# B&R Automation Studio project AutomatedPongGame (part 3)

#### testSet_FieldMotor_Disabled.c
```c
/********************************************************************
 * COPYRIGHT - MyAutoMation-IT
 ********************************************************************
 * Author: Raivo Berends
 ********************************************************************/

#include <bur/plctypes.h>

#ifdef _DEFAULT_INCLUDES
#include <AsDefault.h>
#endif

#include "UnitTest.h"
#include "Library.h"
#include "CommonTypes.h"
#include <string.h>

_SETUP_TEST(void)
{
	FieldMotorFB.FieldMotor = &FieldMotorStruct;
	memset(	FieldMotorFB.FieldMotor, 0, sizeof(*FieldMotorFB.FieldMotor));
	FieldMotorFB.FieldMotor->STS.StateInt = STATE_DISABLED;

	TEST_DONE;
}

_TEST test_Disabled_AllOutputsOff(void)
{
	FB_FieldMotor(&FieldMotorFB);

	TEST_ASSERT_EQUAL_INT(0, FieldMotorFB.FieldMotor->CS.Power);
	TEST_ASSERT_EQUAL_INT(0, FieldMotorFB.FieldMotor->CS.Home);
	TEST_ASSERT_EQUAL_INT(0, FieldMotorFB.FieldMotor->CS.MoveJogNeg);
	TEST_ASSERT_EQUAL_INT(0, FieldMotorFB.FieldMotor->CS.MoveJogPos);
	TEST_ASSERT_EQUAL_INT(0, FieldMotorFB.FieldMotor->CS.MoveAbsolute);

	TEST_DONE;
}

_TEST test_Disabled_StatusFlags(void)
{
	FB_FieldMotor(&FieldMotorFB);

	TEST_ASSERT_EQUAL_INT(1, FieldMotorFB.FieldMotor->STS.Disabled);
	TEST_ASSERT_EQUAL_INT(0, FieldMotorFB.FieldMotor->STS.Initializing);
	TEST_ASSERT_EQUAL_INT(0, FieldMotorFB.FieldMotor->STS.Running);
	TEST_ASSERT_EQUAL_INT(0, FieldMotorFB.FieldMotor->STS.Idle);

	TEST_DONE;
}

_TEST test_Disabled_InternalStateReset(void)
{
	FB_FieldMotor(&FieldMotorFB);

	TEST_ASSERT_EQUAL_INT(0, FieldMotorFB.FieldMotor->STS.EndButtonHit);
	TEST_ASSERT_EQUAL_INT(0, FieldMotorFB.FieldMotor->STS.TimerStarted);
	TEST_ASSERT_EQUAL_INT(0, FieldMotorFB.FieldMotor->STS.TimerEnded);
	TEST_ASSERT_EQUAL_INT(0, FieldMotorFB.FieldMotor->STS.ReferencePosition);
	TEST_ASSERT_EQUAL_INT(0, FieldMotorFB.FieldMotor->STS.AtTargetPosition);

	TEST_DONE;
}

_TEST test_Disabled_NoTransitionWithoutInit(void)
{
	FieldMotorFB.FieldMotor->CS.Initialize = 0;

	FB_FieldMotor(&FieldMotorFB);

	TEST_ASSERT_EQUAL_INT(STATE_DISABLED, FieldMotorFB.FieldMotor->STS.StateInt);

	TEST_DONE;
}

_TEST test_Disabled_TransitionsToInitializing(void)
{
	FieldMotorFB.FieldMotor->CS.Initialize = 1;
	FieldMotorFB.FieldMotor->STS.AlarmActive = 0;
	FieldMotorFB.FieldMotor->STS.Interlocked = 0;

	FB_FieldMotor(&FieldMotorFB);

	TEST_ASSERT_EQUAL_INT(STATE_INITIALIZING, FieldMotorFB.FieldMotor->STS.StateInt);

	TEST_DONE;
}

_TEST test_Disabled_BlockedByAlarm(void)
{
	FieldMotorFB.FieldMotor->CS.Initialize = 1;
	FieldMotorFB.FieldMotor->STS.AlarmActive = 1;

	FB_FieldMotor(&FieldMotorFB);

	TEST_ASSERT_EQUAL_INT(STATE_DISABLED, FieldMotorFB.FieldMotor->STS.StateInt);

	TEST_DONE;
}

_TEST test_Disabled_BlockedByInterlock(void)
{
	FieldMotorFB.FieldMotor->CS.Initialize = 1;
	FieldMotorFB.FieldMotor->STS.Interlocked = 1;

	FB_FieldMotor(&FieldMotorFB);

	TEST_ASSERT_EQUAL_INT(STATE_DISABLED, FieldMotorFB.FieldMotor->STS.StateInt);

	TEST_DONE;
}
/*
B+R UnitTest: This is generated code.
Do not edit! Do not move!
Description: UnitTest Testprogramm infrastructure (TestSet).
LastUpdated: 2026-05-01 12:38:40Z
By B+R UnitTest Helper Version: 2.0.2.35
*/
UNITTEST_FIXTURES(fixtures)
{
	new_TestFixture("test_Disabled_AllOutputsOff", test_Disabled_AllOutputsOff),
	new_TestFixture("test_Disabled_StatusFlags", test_Disabled_StatusFlags),
	new_TestFixture("test_Disabled_InternalStateReset", test_Disabled_InternalStateReset),
	new_TestFixture("test_Disabled_NoTransitionWithoutInit", test_Disabled_NoTransitionWithoutInit),
	new_TestFixture("test_Disabled_TransitionsToInitializing", test_Disabled_TransitionsToInitializing),
	new_TestFixture("test_Disabled_BlockedByAlarm", test_Disabled_BlockedByAlarm),
	new_TestFixture("test_Disabled_BlockedByInterlock", test_Disabled_BlockedByInterlock),
};

UNITTEST_CALLER_COMPLETE_EXPLICIT(testSet_FieldMotor_Disabled, "testSet_FieldMotor_Disabled", setupTest, 0, fixtures, 0, 0, 0);
```

#### testSet_FieldMotor_Initializing.c
```c
/********************************************************************
 * COPYRIGHT - MyAutoMation-IT
 ********************************************************************
 * Author: Raivo Berends
 ********************************************************************/

#include <bur/plctypes.h>

#ifdef _DEFAULT_INCLUDES
#include <AsDefault.h>
#endif

#include "UnitTest.h"
#include "Library.h"
#include "CommonTypes.h"
#include <string.h>

#define ENDBUTTON_BITMASK 0x4

_SETUP_TEST(void)
{
	FieldMotorFB.FieldMotor = &FieldMotorStruct;
	memset(FieldMotorFB.FieldMotor, 0, sizeof(*FieldMotorFB.FieldMotor));
	FieldMotorFB.digitalInput = 0;
	FieldMotorFB.FieldMotor->STS.StateInt = STATE_INITIALIZING;

	TEST_DONE;
}

_TEST test_Initializing_SetsPowerAndParameters(void)
{
	FB_FieldMotor(&FieldMotorFB);

	TEST_ASSERT_EQUAL_INT(1, FieldMotorFB.FieldMotor->CS.Power);
	TEST_ASSERT_EQUAL_INT(0, FieldMotorFB.FieldMotor->CS.Stop);

	TEST_ASSERT_EQUAL_INT(MAX_ACC_DEC, FieldMotorFB.FieldMotor->PAR.Acceleration);
	TEST_ASSERT_EQUAL_INT(MAX_ACC_DEC, FieldMotorFB.FieldMotor->PAR.Deceleration);

	TEST_DONE;
}

_TEST test_Initializing_StartsHomingSequence(void)
{
	FieldMotorFB.digitalInput = ENDBUTTON_BITMASK;
	FieldMotorFB.FieldMotor->STS.EndButtonHit = 0;

	FB_FieldMotor(&FieldMotorFB);

	TEST_ASSERT_EQUAL_INT(1, FieldMotorFB.FieldMotor->CS.Home);
	TEST_ASSERT_EQUAL_INT(1, FieldMotorFB.FieldMotor->STS.TimerStarted);

	TEST_DONE;
}

_TEST test_Initializing_EndButtonHit_TriggersCentering(void)
{
	FieldMotorFB.digitalInput = 0;
	FieldMotorFB.FieldMotor->STS.EndButtonHit = 0;

	FB_FieldMotor(&FieldMotorFB);

	TEST_ASSERT_EQUAL_INT(1, FieldMotorFB.FieldMotor->STS.EndButtonHit);
	TEST_ASSERT_EQUAL_INT(1, FieldMotorFB.FieldMotor->CS.Home);
	TEST_ASSERT_EQUAL_INT(1, FieldMotorFB.FieldMotor->CS.SetCenterPoint);

	TEST_DONE;
}

_TEST test_Initializing_TransitionsToIdle(void)
{
	FieldMotorFB.FieldMotor->STS.EndButtonHit = 1;
	FieldMotorFB.FieldMotor->STS.AtTargetPosition = 1;

	FB_FieldMotor(&FieldMotorFB);

	TEST_ASSERT_EQUAL_INT(STATE_IDLE, FieldMotorFB.FieldMotor->STS.StateInt);

	TEST_DONE;
}

_TEST test_Initializing_BlockedByAlarm(void)
{
	FieldMotorFB.FieldMotor->STS.EndButtonHit = 1;
	FieldMotorFB.FieldMotor->STS.AtTargetPosition = 1;
	FieldMotorFB.FieldMotor->STS.AlarmActive = 1;

	FB_FieldMotor(&FieldMotorFB);

	TEST_ASSERT_EQUAL_INT(STATE_INITIALIZING, FieldMotorFB.FieldMotor->STS.StateInt);

	TEST_DONE;
}

_TEST test_Initializing_BlockedByInterlock(void)
{
	FieldMotorFB.FieldMotor->STS.EndButtonHit = 1;
	FieldMotorFB.FieldMotor->STS.AtTargetPosition = 1;
	FieldMotorFB.FieldMotor->STS.Interlocked = 1;

	FB_FieldMotor(&FieldMotorFB);

	TEST_ASSERT_EQUAL_INT(STATE_INITIALIZING, FieldMotorFB.FieldMotor->STS.StateInt);

	TEST_DONE;
}
/*
B+R UnitTest: This is generated code.
Do not edit! Do not move!
Description: UnitTest Testprogramm infrastructure (TestSet).
LastUpdated: 2026-05-01 13:01:47Z
By B+R UnitTest Helper Version: 2.0.2.35
*/
UNITTEST_FIXTURES(fixtures)
{
	new_TestFixture("test_Initializing_SetsPowerAndParameters", test_Initializing_SetsPowerAndParameters),
	new_TestFixture("test_Initializing_StartsHomingSequence", test_Initializing_StartsHomingSequence),
	new_TestFixture("test_Initializing_EndButtonHit_TriggersCentering", test_Initializing_EndButtonHit_TriggersCentering),
	new_TestFixture("test_Initializing_TransitionsToIdle", test_Initializing_TransitionsToIdle),
	new_TestFixture("test_Initializing_BlockedByAlarm", test_Initializing_BlockedByAlarm),
	new_TestFixture("test_Initializing_BlockedByInterlock", test_Initializing_BlockedByInterlock),
};

UNITTEST_CALLER_COMPLETE_EXPLICIT(testSet_FieldMotor_Initializing, "testSet_FieldMotor_Initializing", setupTest, 0, fixtures, 0, 0, 0);
```

#### testSet_FieldMotor_Idle.c
```c
/********************************************************************
 * COPYRIGHT - MyAutoMation-IT
 ********************************************************************
 * Author: Raivo Berends
 ********************************************************************/

#include <bur/plctypes.h>

#ifdef _DEFAULT_INCLUDES
#include <AsDefault.h>
#endif

#include "UnitTest.h"
#include "Library.h"
#include "CommonTypes.h"
#include <string.h>

_SETUP_TEST(void)
{
	FieldMotorFB.FieldMotor = &FieldMotorStruct;
	memset(	FieldMotorFB.FieldMotor, 0, sizeof(*FieldMotorFB.FieldMotor));
	FieldMotorFB.FieldMotor->STS.StateInt = STATE_IDLE;

	TEST_DONE;
}

_TEST test_Idle_AllOutputsOff(void)
{
	FB_FieldMotor(&FieldMotorFB);

	TEST_ASSERT_EQUAL_INT(0, FieldMotorFB.FieldMotor->CS.MoveAbsolute);
	TEST_ASSERT_EQUAL_INT(0, FieldMotorFB.FieldMotor->CS.MoveJogNeg);
	TEST_ASSERT_EQUAL_INT(0, FieldMotorFB.FieldMotor->CS.MoveJogPos);
	TEST_ASSERT_EQUAL_INT(0, FieldMotorFB.FieldMotor->CS.Power);

	TEST_DONE;
}

_TEST test_Idle_StatusFlags(void)
{
	FB_FieldMotor(&FieldMotorFB);

	TEST_ASSERT_EQUAL_INT(1, FieldMotorFB.FieldMotor->STS.Idle);
	TEST_ASSERT_EQUAL_INT(0, FieldMotorFB.FieldMotor->STS.Initializing);
	TEST_ASSERT_EQUAL_INT(0, FieldMotorFB.FieldMotor->STS.Running);

	TEST_DONE;
}

_TEST test_Idle_NoTransitionWithoutStart(void)
{
	FieldMotorFB.FieldMotor->CS.Start = 0;

	FB_FieldMotor(&FieldMotorFB);

	TEST_ASSERT_EQUAL_INT(STATE_IDLE, FieldMotorFB.FieldMotor->STS.StateInt);

	TEST_DONE;
}

_TEST test_Idle_TransitionToRunning(void)
{
	FieldMotorFB.FieldMotor->CS.Start = 1;

	FB_FieldMotor(&FieldMotorFB);

	TEST_ASSERT_EQUAL_INT(STATE_RUNNING, FieldMotorFB.FieldMotor->STS.StateInt);

	TEST_DONE;
}

_TEST test_Idle_BlockedByAlarm(void)
{
	FieldMotorFB.FieldMotor->CS.Start = 1;
	FieldMotorFB.FieldMotor->STS.AlarmActive = 1;

	FB_FieldMotor(&FieldMotorFB);

	TEST_ASSERT_EQUAL_INT(STATE_IDLE, FieldMotorFB.FieldMotor->STS.StateInt);

	TEST_DONE;
}

_TEST test_Idle_BlockedByInterlock(void)
{
	FieldMotorFB.FieldMotor->CS.Start = 1;
	FieldMotorFB.FieldMotor->STS.Interlocked = 1;

	FB_FieldMotor(&FieldMotorFB);

	TEST_ASSERT_EQUAL_INT(STATE_IDLE, FieldMotorFB.FieldMotor->STS.StateInt);

	TEST_DONE;
}
/*
B+R UnitTest: This is generated code.
Do not edit! Do not move!
Description: UnitTest Testprogramm infrastructure (TestSet).
LastUpdated: 2026-05-07 09:05:51Z
By B+R UnitTest Helper Version: 2.0.2.35
*/
UNITTEST_FIXTURES(fixtures)
{
	new_TestFixture("test_Idle_AllOutputsOff", test_Idle_AllOutputsOff),
	new_TestFixture("test_Idle_StatusFlags", test_Idle_StatusFlags),
	new_TestFixture("test_Idle_NoTransitionWithoutStart", test_Idle_NoTransitionWithoutStart),
	new_TestFixture("test_Idle_TransitionToRunning", test_Idle_TransitionToRunning),
	new_TestFixture("test_Idle_BlockedByAlarm", test_Idle_BlockedByAlarm),
	new_TestFixture("test_Idle_BlockedByInterlock", test_Idle_BlockedByInterlock),
};

UNITTEST_CALLER_COMPLETE_EXPLICIT(testSet_FieldMotor_Idle, "testSet_FieldMotor_Idle", setupTest, 0, fixtures, 0, 0, 0);
```

#### testSet_FieldMotor_Running.c
```c
/********************************************************************
 * COPYRIGHT - MyAutoMation-IT
 ********************************************************************
 * Author: Raivo Berends
 ********************************************************************/

#include <bur/plctypes.h>

#ifdef _DEFAULT_INCLUDES
#include <AsDefault.h>
#endif

#include "UnitTest.h"
#include "Library.h"
#include "CommonTypes.h"
#include <string.h>

_SETUP_TEST(void)
{
	FieldMotorFB.FieldMotor = &FieldMotorStruct;
	memset(	FieldMotorFB.FieldMotor, 0, sizeof(*FieldMotorFB.FieldMotor));
	FieldMotorFB.FieldMotor->STS.StateInt = STATE_RUNNING;

	TEST_DONE;
}

_TEST Test_Running_SetsRunningAndPower(void)
{
	FB_FieldMotor(&FieldMotorFB);

	TEST_ASSERT_EQUAL_INT(1, FieldMotorFB.FieldMotor->STS.Running);
	TEST_ASSERT_EQUAL_INT(1, FieldMotorFB.FieldMotor->CS.Power);
	TEST_ASSERT_EQUAL_INT(0, FieldMotorFB.FieldMotor->STS.Idle);

	TEST_DONE;
}

_TEST Test_Running_ResetsMovementCommands(void)
{
	FieldMotorFB.FieldMotor->STS.AutoActive = 0;

	FieldMotorFB.FieldMotor->CS.MoveAbsolute = 1;
	FieldMotorFB.FieldMotor->CS.MoveJogNeg = 1;
	FieldMotorFB.FieldMotor->CS.MoveJogPos = 1;

	FB_FieldMotor(&FieldMotorFB);

	TEST_ASSERT_EQUAL_INT(0, FieldMotorFB.FieldMotor->CS.MoveAbsolute);
	TEST_ASSERT_EQUAL_INT(0, FieldMotorFB.FieldMotor->CS.MoveJogNeg);
	TEST_ASSERT_EQUAL_INT(0, FieldMotorFB.FieldMotor->CS.MoveJogPos);

	TEST_DONE;
}

_TEST Test_Running_IncreaseJogSpeed(void)
{
	FieldMotorFB.FieldMotor->STS.AutoActive = 0;

	FieldMotorFB.FieldMotor->PAR.JogVelocity = 10;
	FieldMotorFB.FieldMotor->HMI.IncreaseJogSpeed = 1;

	FB_FieldMotor(&FieldMotorFB);

	TEST_ASSERT_EQUAL_INT(11, FieldMotorFB.FieldMotor->PAR.JogVelocity);

	TEST_DONE;
}

_TEST Test_Running_MaxJogSpeedLimit(void)
{
	FieldMotorFB.FieldMotor->STS.AutoActive = 0;

	FieldMotorFB.FieldMotor->PAR.JogVelocity = MAX_VELOCITY;
	FieldMotorFB.FieldMotor->HMI.IncreaseJogSpeed = 1;

	FB_FieldMotor(&FieldMotorFB);

	TEST_ASSERT_EQUAL_INT(MAX_VELOCITY, FieldMotorFB.FieldMotor->PAR.JogVelocity);

	TEST_DONE;
}

_TEST Test_Running_DecreaseJogSpeed(void)
{
	FieldMotorFB.FieldMotor->STS.AutoActive = 0;

	FieldMotorFB.FieldMotor->PAR.JogVelocity = 1000;
	FieldMotorFB.FieldMotor->HMI.DecreaseJogSpeed = 1;

	FB_FieldMotor(&FieldMotorFB);

	TEST_ASSERT_EQUAL_INT(999, FieldMotorFB.FieldMotor->PAR.JogVelocity);

	TEST_DONE;
}

_TEST Test_Running_MinJogSpeedLimit(void)
{
	FieldMotorFB.FieldMotor->STS.AutoActive = 0;

	FieldMotorFB.FieldMotor->PAR.JogVelocity = MIN_VELOCITY;
	FieldMotorFB.FieldMotor->HMI.DecreaseJogSpeed = 1;

	FB_FieldMotor(&FieldMotorFB);

	TEST_ASSERT_EQUAL_INT(MIN_VELOCITY, FieldMotorFB.FieldMotor->PAR.JogVelocity);

	TEST_DONE;
}

_TEST Test_Running_EndButtonStopsPositiveMovement(void)
{
	FieldMotorFB.digitalInput = !ENDBUTTON_BITMASK_FIELD;

	FieldMotorFB.FieldMotor->CS.MoveJogPos = 1;
	FieldMotorFB.FieldMotor->HMI.MoveJogPos = 1;
	FieldMotorFB.FieldMotor->CS.MoveAbsolute = 1;

	FB_FieldMotor(&FieldMotorFB);

	TEST_ASSERT_EQUAL_INT(0, FieldMotorFB.FieldMotor->CS.MoveJogPos);
	TEST_ASSERT_EQUAL_INT(0, FieldMotorFB.FieldMotor->HMI.MoveJogPos);
	TEST_ASSERT_EQUAL_INT(0, FieldMotorFB.FieldMotor->CS.MoveAbsolute);

	TEST_DONE;
}

_TEST Test_Running_StopGameTransitionsToStopping(void)
{
	FieldMotorFB.FieldMotor->CS.StopGame = 1;
	FieldMotorFB.FieldMotor->STS.AlarmActive = 0;
	FieldMotorFB.FieldMotor->STS.Interlocked = 0;

	FB_FieldMotor(&FieldMotorFB);

	TEST_ASSERT_EQUAL_INT(STATE_STOPPING, FieldMotorFB.FieldMotor->STS.StateInt);

	TEST_DONE;
}

_TEST Test_Running_StopBlockedByInterlock(void)
{
	FieldMotorFB.FieldMotor->CS.StopGame = 1;
	FieldMotorFB.FieldMotor->STS.Interlocked = 1;

	FB_FieldMotor(&FieldMotorFB);

	TEST_ASSERT_EQUAL_INT(STATE_RUNNING, FieldMotorFB.FieldMotor->STS.StateInt);

	TEST_DONE;
}

_TEST Test_Running_StandStillDetection(void)
{
	FieldMotorFB.FieldMotor->STS.ActVelocity = 0;

	FB_FieldMotor(&FieldMotorFB);

	TEST_ASSERT_EQUAL_INT(1, FieldMotorFB.FieldMotor->STS.StandStill);
	TEST_ASSERT_EQUAL_INT(0, FieldMotorFB.FieldMotor->STS.Moving);

	TEST_DONE;
}

_TEST Test_Running_MovingDetection(void)
{
	FieldMotorFB.FieldMotor->STS.ActVelocity = 100;

	FB_FieldMotor(&FieldMotorFB);

	TEST_ASSERT_EQUAL_INT(0, FieldMotorFB.FieldMotor->STS.StandStill);
	TEST_ASSERT_EQUAL_INT(1, FieldMotorFB.FieldMotor->STS.Moving);

	TEST_DONE;
}

_TEST Test_Running_XorMoveJogPos(void)
{
	FieldMotorFB.FieldMotor->CS.MoveJogPos = 0;
	FieldMotorFB.FieldMotor->HMI.MoveJogPos = 1;
	FieldMotorFB.digitalInput = ENDBUTTON_BITMASK_FIELD;

	FB_FieldMotor(&FieldMotorFB);

	TEST_ASSERT_EQUAL_INT(1, FieldMotorFB.FieldMotor->IO.MoveJogPos);

	TEST_DONE;
}

_TEST Test_Running_XorMoveJogPosBothHigh(void)
{
	FieldMotorFB.FieldMotor->CS.MoveJogPos = 1;
	FieldMotorFB.FieldMotor->HMI.MoveJogPos = 1;
	FieldMotorFB.digitalInput = ENDBUTTON_BITMASK_FIELD;

	FB_FieldMotor(&FieldMotorFB);

	TEST_ASSERT_EQUAL_INT(1, FieldMotorFB.FieldMotor->IO.MoveJogPos);

	TEST_DONE;
}

_TEST Test_Running_AlarmSourcePropagation(void)
{
	FieldMotorFB.FieldMotor->ALM.MotorError = 1;

	FB_FieldMotor(&FieldMotorFB);

	TEST_ASSERT_EQUAL_INT(1, FieldMotorFB.FieldMotor->STS.AlarmActive);

	TEST_DONE;
}

/*
B+R UnitTest: This is generated code.
Do not edit! Do not move!
Description: UnitTest Testprogramm infrastructure (TestSet).
LastUpdated: 2026-05-19 08:31:48Z
By B+R UnitTest Helper Version: 2.0.2.35
*/
UNITTEST_FIXTURES(fixtures)
{
	new_TestFixture("Test_Running_SetsRunningAndPower", Test_Running_SetsRunningAndPower),
	new_TestFixture("Test_Running_ResetsMovementCommands", Test_Running_ResetsMovementCommands),
	new_TestFixture("Test_Running_IncreaseJogSpeed", Test_Running_IncreaseJogSpeed),
	new_TestFixture("Test_Running_MaxJogSpeedLimit", Test_Running_MaxJogSpeedLimit),
	new_TestFixture("Test_Running_DecreaseJogSpeed", Test_Running_DecreaseJogSpeed),
	new_TestFixture("Test_Running_MinJogSpeedLimit", Test_Running_MinJogSpeedLimit),
	new_TestFixture("Test_Running_EndButtonStopsPositiveMovement", Test_Running_EndButtonStopsPositiveMovement),
	new_TestFixture("Test_Running_StopGameTransitionsToStopping", Test_Running_StopGameTransitionsToStopping),
	new_TestFixture("Test_Running_StopBlockedByInterlock", Test_Running_StopBlockedByInterlock),
	new_TestFixture("Test_Running_StandStillDetection", Test_Running_StandStillDetection),
	new_TestFixture("Test_Running_MovingDetection", Test_Running_MovingDetection),
	new_TestFixture("Test_Running_XorMoveJogPos", Test_Running_XorMoveJogPos),
	new_TestFixture("Test_Running_XorMoveJogPosBothHigh", Test_Running_XorMoveJogPosBothHigh),
	new_TestFixture("Test_Running_AlarmSourcePropagation", Test_Running_AlarmSourcePropagation),
};

UNITTEST_CALLER_COMPLETE_EXPLICIT(testSet_FieldMotor_Running, "testSet_FieldMotor_Running", setupTest, 0, fixtures, 0, 0, 0);
```

#### testSet_FieldMotor_Stopping.c
```c
/********************************************************************
 * COPYRIGHT - MyAutoMation-IT
 ********************************************************************
 * Author: Raivo Berends
 ********************************************************************/

#include <bur/plctypes.h>

#ifdef _DEFAULT_INCLUDES
#include <AsDefault.h>
#endif

#include "UnitTest.h"
#include "Library.h"
#include "CommonTypes.h"
#include <string.h>

_SETUP_TEST(void)
{
	FieldMotorFB.FieldMotor = &FieldMotorStruct;
	memset(	FieldMotorFB.FieldMotor, 0, sizeof(*FieldMotorFB.FieldMotor));
	FieldMotorFB.FieldMotor->STS.StateInt = STATE_IDLE;

	TEST_DONE;
}

_TEST Test_Stopping_ResetsStateFlags(void)
{
	FieldMotorFB.FieldMotor->STS.StateInt = STATE_STOPPING;

	FieldMotorFB.FieldMotor->STS.Running = 1;
	FieldMotorFB.FieldMotor->STS.Idle = 1;
	FieldMotorFB.FieldMotor->STS.Initializing = 1;

	FB_FieldMotor(&FieldMotorFB);

	TEST_ASSERT_EQUAL_INT(0, FieldMotorFB.FieldMotor->STS.Running);
	TEST_ASSERT_EQUAL_INT(0, FieldMotorFB.FieldMotor->STS.Idle);
	TEST_ASSERT_EQUAL_INT(0, FieldMotorFB.FieldMotor->STS.Initializing);

	TEST_DONE;
}

_TEST Test_Stopping_StopsAllMovement(void)
{
	FieldMotorFB.FieldMotor->STS.StateInt = STATE_STOPPING;

	FieldMotorFB.FieldMotor->CS.MoveAbsolute = 1;
	FieldMotorFB.FieldMotor->CS.MoveJogNeg = 1;
	FieldMotorFB.FieldMotor->CS.MoveJogPos = 1;

	FB_FieldMotor(&FieldMotorFB);

	TEST_ASSERT_EQUAL_INT(0, FieldMotorFB.FieldMotor->CS.MoveAbsolute);
	TEST_ASSERT_EQUAL_INT(0, FieldMotorFB.FieldMotor->CS.MoveJogNeg);
	TEST_ASSERT_EQUAL_INT(0, FieldMotorFB.FieldMotor->CS.MoveJogPos);

	TEST_DONE;
}

_TEST Test_Stopping_SetsStopCommand(void)
{
	FieldMotorFB.FieldMotor->STS.StateInt = STATE_STOPPING;

	FieldMotorFB.FieldMotor->CS.Stop = 0;

	FB_FieldMotor(&FieldMotorFB);

	TEST_ASSERT_EQUAL_INT(1, FieldMotorFB.FieldMotor->CS.Stop);

	TEST_DONE;
}

_TEST Test_Stopping_TransitionsToDisabled(void)
{
	FieldMotorFB.FieldMotor->STS.StateInt = STATE_STOPPING;

	FieldMotorFB.FieldMotor->STS.StandStill = 1;
	FieldMotorFB.FieldMotor->STS.Interlocked = 0;

	FB_FieldMotor(&FieldMotorFB);

	TEST_ASSERT_EQUAL_INT(STATE_DISABLED, FieldMotorFB.FieldMotor->STS.StateInt);

	TEST_DONE;
}

_TEST Test_Stopping_DoesNotTransitionWhenMoving(void)
{
	FieldMotorFB.FieldMotor->STS.StateInt = STATE_STOPPING;

	FieldMotorFB.FieldMotor->STS.StandStill = 0;
	FieldMotorFB.FieldMotor->STS.Interlocked = 0;

	FB_FieldMotor(&FieldMotorFB);

	TEST_ASSERT_EQUAL_INT(STATE_STOPPING, FieldMotorFB.FieldMotor->STS.StateInt);

	TEST_DONE;
}

_TEST Test_Stopping_DoesNotTransitionWhenInterlocked(void)
{
	FieldMotorFB.FieldMotor->STS.StateInt = STATE_STOPPING;

	FieldMotorFB.FieldMotor->STS.StandStill = 1;
	FieldMotorFB.FieldMotor->STS.Interlocked = 1;

	FB_FieldMotor(&FieldMotorFB);

	TEST_ASSERT_EQUAL_INT(STATE_STOPPING, FieldMotorFB.FieldMotor->STS.StateInt);

	TEST_DONE;
}

_TEST Test_Stopping_UpdatesStopOutput(void)
{
	FieldMotorFB.FieldMotor->STS.StateInt = STATE_STOPPING;

	FB_FieldMotor(&FieldMotorFB);

	TEST_ASSERT_EQUAL_INT(1, FieldMotorFB.FieldMotor->IO.Stop);

	TEST_DONE;
}

/*
B+R UnitTest: This is generated code.
Do not edit! Do not move!
Description: UnitTest Testprogramm infrastructure (TestSet).
LastUpdated: 2026-05-07 09:05:51Z
By B+R UnitTest Helper Version: 2.0.2.35
*/
UNITTEST_FIXTURES(fixtures)
{
	new_TestFixture("Test_Stopping_ResetsStateFlags", Test_Stopping_ResetsStateFlags),
	new_TestFixture("Test_Stopping_StopsAllMovement", Test_Stopping_StopsAllMovement),
	new_TestFixture("Test_Stopping_SetsStopCommand", Test_Stopping_SetsStopCommand),
	new_TestFixture("Test_Stopping_TransitionsToDisabled", Test_Stopping_TransitionsToDisabled),
	new_TestFixture("Test_Stopping_DoesNotTransitionWhenMoving", Test_Stopping_DoesNotTransitionWhenMoving),
	new_TestFixture("Test_Stopping_DoesNotTransitionWhenInterlocked", Test_Stopping_DoesNotTransitionWhenInterlocked),
	new_TestFixture("Test_Stopping_UpdatesStopOutput", Test_Stopping_UpdatesStopOutput),
};

UNITTEST_CALLER_COMPLETE_EXPLICIT(testSet_FieldMotor_Stopping, "testSet_FieldMotor_Stopping", setupTest, 0, fixtures, 0, 0, 0);
```

### Program Logical/UnitTests/UnitTests/Tests_PaddleMotor_C (ANSIC) - Empty template for use with helper tool

#### autoGeneratedFile.c
```c
/*
B+R UnitTest: This is generated code.
Do not edit! Do not move!
Description: UnitTest Testprogramm infrastructure (List of TestSets).
LastUpdated: 2026-05-01 12:04:37Z
By B+R UnitTest Helper Version: 2.0.2.35
*/
#include "UnitTest.h"

UNITTEST_TESTSET_DECLARATION  testSet_PaddleMotor_Disabled;
UNITTEST_TESTSET_DECLARATION  testSet_PaddleMotor_Initializing;
UNITTEST_TESTSET_DECLARATION  testSet_PaddleMotor_Idle;
UNITTEST_TESTSET_DECLARATION  testSet_PaddleMotor_Running;
UNITTEST_TESTSET_DECLARATION  testSet_PaddleMotor_Stopping;

UNITTEST_TESTSET_FIXTURES(utTestSets)
{
	new_TestSet(testSet_PaddleMotor_Disabled),
	new_TestSet(testSet_PaddleMotor_Initializing),
	new_TestSet(testSet_PaddleMotor_Idle),
	new_TestSet(testSet_PaddleMotor_Running),
	new_TestSet(testSet_PaddleMotor_Stopping),
};
UNTITTEST_TESTSET_HANDLER();
```

#### testSet_PaddleMotor_Disabled.c
```c
/********************************************************************
 * COPYRIGHT - MyAutoMation-IT
 ********************************************************************
 * Author: Raivo Berends
 ********************************************************************/

#include <bur/plctypes.h>

#ifdef _DEFAULT_INCLUDES
#include <AsDefault.h>
#endif

#include "UnitTest.h"
#include "Library.h"
#include "CommonTypes.h"
#include <string.h>

_SETUP_TEST(void)
{
	/* TODO:  add code running before test set here */
	PaddleMotorFB.PaddleMotor = &PaddleMotorStruct;
	memset(PaddleMotorFB.PaddleMotor, 0, sizeof(*PaddleMotorFB.PaddleMotor));
	PaddleMotorFB.PaddleMotor->STS.StateInt = STATE_DISABLED;

	TEST_DONE;
}

_TEST test_Disabled_State_DefaultBehavior(void)
{
	PaddleMotorFB.digitalInput = 0;

	// Setting signals that have to be reset
	PaddleMotorFB.PaddleMotor->CS.Power = 1;
	PaddleMotorFB.PaddleMotor->CS.Home = 1;
	PaddleMotorFB.PaddleMotor->CS.MoveJogNeg = 1;
	PaddleMotorFB.PaddleMotor->CS.MoveJogPos = 1;
	PaddleMotorFB.PaddleMotor->CS.MoveAbsolute = 1;

	PaddleMotorFB.PaddleMotor->HMI.MoveJogNeg = 1;
	PaddleMotorFB.PaddleMotor->HMI.MoveJogPos = 1;

	PaddleMotorFB.PaddleMotor->STS.TimerStarted = 1;
	PaddleMotorFB.PaddleMotor->STS.TimerEnded = 1;
	PaddleMotorFB.PaddleMotor->STS.ReferencePosition = 1234;
	PaddleMotorFB.PaddleMotor->STS.ReferenceSet = 1;

	FB_PaddleMotor(&PaddleMotorFB);

	TEST_ASSERT_EQUAL_INT(1, PaddleMotorFB.PaddleMotor->STS.Disabled);

	TEST_ASSERT_EQUAL_INT(0, PaddleMotorFB.PaddleMotor->CS.Power);
	TEST_ASSERT_EQUAL_INT(0, PaddleMotorFB.PaddleMotor->CS.Home);
	TEST_ASSERT_EQUAL_INT(0, PaddleMotorFB.PaddleMotor->CS.MoveJogNeg);
	TEST_ASSERT_EQUAL_INT(0, PaddleMotorFB.PaddleMotor->CS.MoveJogPos);
	TEST_ASSERT_EQUAL_INT(0, PaddleMotorFB.PaddleMotor->CS.MoveAbsolute);

	TEST_ASSERT_EQUAL_INT(0, PaddleMotorFB.PaddleMotor->HMI.MoveJogNeg);
	TEST_ASSERT_EQUAL_INT(0, PaddleMotorFB.PaddleMotor->HMI.MoveJogPos);

	TEST_ASSERT_EQUAL_INT(0, PaddleMotorFB.PaddleMotor->STS.TimerStarted);
	TEST_ASSERT_EQUAL_INT(0, PaddleMotorFB.PaddleMotor->STS.TimerEnded);
	TEST_ASSERT_EQUAL_INT(0, PaddleMotorFB.PaddleMotor->STS.ReferencePosition);
	TEST_ASSERT_EQUAL_INT(0, PaddleMotorFB.PaddleMotor->STS.ReferenceSet);

	TEST_DONE;
}

_TEST test_Disabled_NoInitialize_StaysDisabled(void)
{
	PaddleMotorFB.PaddleMotor->CS.Initialize = 0;
	PaddleMotorFB.PaddleMotor->STS.AlarmActive = 0;
	PaddleMotorFB.PaddleMotor->STS.Interlocked = 0;

	FB_PaddleMotor(&PaddleMotorFB);

	TEST_ASSERT_EQUAL_INT(STATE_DISABLED, PaddleMotorFB.PaddleMotor->STS.StateInt);

	TEST_DONE;
}

_TEST test_Disabled_ToInitializing(void)
{
	PaddleMotorFB.PaddleMotor->CS.Initialize = 1;
	PaddleMotorFB.PaddleMotor->STS.AlarmActive = 0;
	PaddleMotorFB.PaddleMotor->STS.Interlocked = 0;

	FB_PaddleMotor(&PaddleMotorFB);

	TEST_ASSERT_EQUAL_INT(STATE_INITIALIZING, PaddleMotorFB.PaddleMotor->STS.StateInt);

	TEST_DONE;
}

_TEST test_Disabled_NoTransition_WhenAlarm(void)
{
	PaddleMotorFB.PaddleMotor->CS.Initialize = 1;
	PaddleMotorFB.PaddleMotor->STS.AlarmActive = 1;
	PaddleMotorFB.PaddleMotor->STS.Interlocked = 0;

	FB_PaddleMotor(&PaddleMotorFB);

	TEST_ASSERT_EQUAL_INT(STATE_DISABLED, PaddleMotorFB.PaddleMotor->STS.StateInt);

	TEST_DONE;
}

_TEST test_Disabled_NoTransition_WhenInterlocked(void)
{
	PaddleMotorFB.PaddleMotor->CS.Initialize = 1;
	PaddleMotorFB.PaddleMotor->STS.AlarmActive = 0;
	PaddleMotorFB.PaddleMotor->STS.Interlocked = 1;

	FB_PaddleMotor(&PaddleMotorFB);

	TEST_ASSERT_EQUAL_INT(STATE_DISABLED, PaddleMotorFB.PaddleMotor->STS.StateInt);

	TEST_DONE;
}

/*
B+R UnitTest: This is generated code.
Do not edit! Do not move!
Description: UnitTest Testprogramm infrastructure (TestSet).
LastUpdated: 2026-04-20 10:39:20Z
By B+R UnitTest Helper Version: 2.0.2.35
*/
UNITTEST_FIXTURES(fixtures)
{
	new_TestFixture("test_Disabled_State_DefaultBehavior", test_Disabled_State_DefaultBehavior),
	new_TestFixture("test_Disabled_NoInitialize_StaysDisabled", test_Disabled_NoInitialize_StaysDisabled),
	new_TestFixture("test_Disabled_ToInitializing", test_Disabled_ToInitializing),
	new_TestFixture("test_Disabled_NoTransition_WhenAlarm", test_Disabled_NoTransition_WhenAlarm),
	new_TestFixture("test_Disabled_NoTransition_WhenInterlocked", test_Disabled_NoTransition_WhenInterlocked),
};

UNITTEST_CALLER_COMPLETE_EXPLICIT(testSet_PaddleMotor_Disabled, "testSet_PaddleMotor_Disabled", setupTest, 0, fixtures, 0, 0, 0);
```

#### testSet_PaddleMotor_Idle.c
```c
/********************************************************************
 * COPYRIGHT - MyAutoMation-IT
 ********************************************************************
 * Author: Raivo Berends
 ********************************************************************/

#include <bur/plctypes.h>

#ifdef _DEFAULT_INCLUDES
#include <AsDefault.h>
#endif

#include "UnitTest.h"
#include "Library.h"
#include "CommonTypes.h"
#include <string.h>

_SETUP_TEST(void)
{
	PaddleMotorFB.PaddleMotor = &PaddleMotorStruct;
	memset(PaddleMotorFB.PaddleMotor, 0, sizeof(*PaddleMotorFB.PaddleMotor));
	PaddleMotorFB.PaddleMotor->STS.StateInt = STATE_IDLE;

	TEST_DONE;
}

_TEST test_Idle_SetsStatusAndResetsOutputs(void)
{
	PaddleMotorFB.PaddleMotor->STS.Initializing = 1;
	PaddleMotorFB.PaddleMotor->STS.Idle = 0;

	PaddleMotorFB.PaddleMotor->CS.MoveAbsolute = 1;
	PaddleMotorFB.PaddleMotor->CS.MoveJogNeg = 1;
	PaddleMotorFB.PaddleMotor->CS.MoveJogPos = 1;

	PaddleMotorFB.PaddleMotor->HMI.MoveAbsolute = 1;
	PaddleMotorFB.PaddleMotor->HMI.MoveJogNeg = 1;
	PaddleMotorFB.PaddleMotor->HMI.MoveJogPos = 1;

	FB_PaddleMotor(&PaddleMotorFB);

	TEST_ASSERT_EQUAL_INT(0, PaddleMotorFB.PaddleMotor->STS.Initializing);
	TEST_ASSERT_EQUAL_INT(1, PaddleMotorFB.PaddleMotor->STS.Idle);

	TEST_ASSERT_EQUAL_INT(0, PaddleMotorFB.PaddleMotor->CS.MoveAbsolute);
	TEST_ASSERT_EQUAL_INT(0, PaddleMotorFB.PaddleMotor->CS.MoveJogNeg);
	TEST_ASSERT_EQUAL_INT(0, PaddleMotorFB.PaddleMotor->CS.MoveJogPos);

	TEST_ASSERT_EQUAL_INT(0, PaddleMotorFB.PaddleMotor->HMI.MoveAbsolute);
	TEST_ASSERT_EQUAL_INT(0, PaddleMotorFB.PaddleMotor->HMI.MoveJogNeg);
	TEST_ASSERT_EQUAL_INT(0, PaddleMotorFB.PaddleMotor->HMI.MoveJogPos);

	TEST_DONE;
}

_TEST test_Idle_RemainsIdleWithoutStart(void)
{
	PaddleMotorFB.PaddleMotor->CS.Start = 0;

	FB_PaddleMotor(&PaddleMotorFB);

	TEST_ASSERT_EQUAL_INT(STATE_IDLE, PaddleMotorFB.PaddleMotor->STS.StateInt);

	TEST_DONE;
}

_TEST test_Idle_ToRunning(void)
{
	PaddleMotorFB.PaddleMotor->CS.Start = 1;
	PaddleMotorFB.PaddleMotor->STS.AlarmActive = 0;
	PaddleMotorFB.PaddleMotor->STS.Interlocked = 0;

	FB_PaddleMotor(&PaddleMotorFB);

	TEST_ASSERT_EQUAL_INT(STATE_RUNNING, PaddleMotorFB.PaddleMotor->STS.StateInt);

	TEST_DONE;
}

_TEST test_Idle_NoTransitionWhenAlarmActive(void)
{
	PaddleMotorFB.PaddleMotor->CS.Start = 1;
	PaddleMotorFB.PaddleMotor->STS.AlarmActive = 1;
	PaddleMotorFB.PaddleMotor->STS.Interlocked = 0;

	FB_PaddleMotor(&PaddleMotorFB);

	TEST_ASSERT_EQUAL_INT(STATE_IDLE, PaddleMotorFB.PaddleMotor->STS.StateInt);

	TEST_DONE;
}

_TEST test_Idle_NoTransitionWhenInterlocked(void)
{
	PaddleMotorFB.PaddleMotor->CS.Start = 1;
	PaddleMotorFB.PaddleMotor->STS.AlarmActive = 0;
	PaddleMotorFB.PaddleMotor->STS.Interlocked = 1;

	FB_PaddleMotor(&PaddleMotorFB);

	TEST_ASSERT_EQUAL_INT(STATE_IDLE, PaddleMotorFB.PaddleMotor->STS.StateInt);

	TEST_DONE;
}

_TEST test_Idle_IOOutputsRemainZero(void)
{
	PaddleMotorFB.PaddleMotor->CS.MoveJogPos = 0;
	PaddleMotorFB.PaddleMotor->HMI.MoveJogPos = 1;

	PaddleMotorFB.PaddleMotor->CS.MoveJogNeg = 0;
	PaddleMotorFB.PaddleMotor->HMI.MoveJogNeg = 1;

	FB_PaddleMotor(&PaddleMotorFB);

	TEST_ASSERT_EQUAL_INT(0, PaddleMotorFB.PaddleMotor->IO.MoveJogPos);
	TEST_ASSERT_EQUAL_INT(0, PaddleMotorFB.PaddleMotor->IO.MoveJogNeg);

	TEST_DONE;
}

/*
B+R UnitTest: This is generated code.
Do not edit! Do not move!
Description: UnitTest Testprogramm infrastructure (TestSet).
LastUpdated: 2026-05-01 11:23:13Z
By B+R UnitTest Helper Version: 2.0.2.35
*/
UNITTEST_FIXTURES(fixtures)
{
	new_TestFixture("test_Idle_SetsStatusAndResetsOutputs", test_Idle_SetsStatusAndResetsOutputs),
	new_TestFixture("test_Idle_RemainsIdleWithoutStart", test_Idle_RemainsIdleWithoutStart),
	new_TestFixture("test_Idle_ToRunning", test_Idle_ToRunning),
	new_TestFixture("test_Idle_NoTransitionWhenAlarmActive", test_Idle_NoTransitionWhenAlarmActive),
	new_TestFixture("test_Idle_NoTransitionWhenInterlocked", test_Idle_NoTransitionWhenInterlocked),
	new_TestFixture("test_Idle_IOOutputsRemainZero", test_Idle_IOOutputsRemainZero),
};

UNITTEST_CALLER_COMPLETE_EXPLICIT(testSet_PaddleMotor_Idle, "testSet_PaddleMotor_Idle", setupTest, 0, fixtures, 0, 0, 0);
```

#### testSet_PaddleMotor_Initializing.c
```c
/********************************************************************
 * COPYRIGHT - MyAutoMation-IT
 ********************************************************************
 * Author: Raivo Berends
 ********************************************************************/

#include <bur/plctypes.h>

#ifdef _DEFAULT_INCLUDES
#include <AsDefault.h>
#endif

#include "UnitTest.h"
#include "Library.h"
#include "CommonTypes.h"
#include <string.h>

#define MIDDLE_POSITION 1450

_SETUP_TEST(void)
{
	PaddleMotorFB.PaddleMotor = &PaddleMotorStruct;
	memset(PaddleMotorFB.PaddleMotor, 0, sizeof(*PaddleMotorFB.PaddleMotor));
	PaddleMotorFB.PaddleMotor->STS.StateInt = STATE_INITIALIZING;

	TEST_DONE;
}

_TEST test_Initializing_SetsParameters(void)
{
	FB_PaddleMotor(&PaddleMotorFB);

	TEST_ASSERT_EQUAL_INT(1, PaddleMotorFB.PaddleMotor->STS.Initializing);
	TEST_ASSERT_EQUAL_INT(0, PaddleMotorFB.PaddleMotor->STS.Disabled);

	TEST_ASSERT_EQUAL_INT(MAX_ACC_DEC, PaddleMotorFB.PaddleMotor->PAR.Acceleration);
	TEST_ASSERT_EQUAL_INT(MAX_ACC_DEC, PaddleMotorFB.PaddleMotor->PAR.Deceleration);
	TEST_ASSERT_EQUAL_INT(1000, PaddleMotorFB.PaddleMotor->PAR.JogVelocity);
	TEST_ASSERT_EQUAL_INT(1000, PaddleMotorFB.PaddleMotor->PAR.Velocity);

	TEST_ASSERT_EQUAL_INT(1, PaddleMotorFB.PaddleMotor->CS.Power);
	TEST_ASSERT_EQUAL_INT(0, PaddleMotorFB.PaddleMotor->CS.Stop);

	TEST_DONE;
}

_TEST test_Initializing_StartsHoming(void)
{
	PaddleMotorFB.digitalInput = ENDBUTTON_BITMASK_PADDLE; // EndButton = inactive

	PaddleMotorFB.PaddleMotor->STS.EndButtonHit = 0;

	FB_PaddleMotor(&PaddleMotorFB);

	TEST_ASSERT_EQUAL_INT(1, PaddleMotorFB.PaddleMotor->CS.Home);
	TEST_ASSERT_EQUAL_INT(1, PaddleMotorFB.PaddleMotor->STS.TimerStarted);

	TEST_DONE;
}

_TEST test_Initializing_EndButtonHit(void)
{
	PaddleMotorFB.digitalInput = 0x1;

	PaddleMotorFB.PaddleMotor->STS.EndButtonHit = 0;

	FB_PaddleMotor(&PaddleMotorFB);

	TEST_ASSERT_EQUAL_INT(1, PaddleMotorFB.PaddleMotor->STS.EndButtonHit);
	TEST_ASSERT_EQUAL_INT(1, PaddleMotorFB.PaddleMotor->CS.Home);
	TEST_ASSERT_EQUAL_INT(0, PaddleMotorFB.PaddleMotor->CS.MoveJogPos);

	TEST_DONE;
}

_TEST test_Initializing_ToIdle(void)
{
	PaddleMotorFB.PaddleMotor->STS.EndButtonHit = 1;
	PaddleMotorFB.PaddleMotor->STS.TimerEnded = 1;
	PaddleMotorFB.PaddleMotor->STS.ReferenceSet = 1;

	PaddleMotorFB.PaddleMotor->PAR.Position = 3000;
	PaddleMotorFB.PaddleMotor->STS.ActPosition = 3000;

	PaddleMotorFB.PaddleMotor->STS.AlarmActive = 0;
	PaddleMotorFB.PaddleMotor->STS.Interlocked = 0;

	FB_PaddleMotor(&PaddleMotorFB);

	TEST_ASSERT_EQUAL_INT(STATE_IDLE, PaddleMotorFB.PaddleMotor->STS.StateInt);
	TEST_ASSERT_EQUAL_INT(0, PaddleMotorFB.PaddleMotor->CS.MoveAbsolute);

	TEST_DONE;
}

_TEST test_Initializing_ReferencePosition(void)
{
	PaddleMotorFB.PaddleMotor->STS.EndButtonHit = 1;
	PaddleMotorFB.PaddleMotor->STS.TimerEnded = 1;
	PaddleMotorFB.PaddleMotor->STS.ReferenceSet = 0;

	PaddleMotorFB.PaddleMotor->STS.ActPosition = 5000;

	FB_PaddleMotor(&PaddleMotorFB);

	TEST_ASSERT_EQUAL_INT(
		PaddleMotorFB.PaddleMotor->STS.ActPosition + 25,
		PaddleMotorFB.PaddleMotor->STS.ReferencePosition
		);

	TEST_DONE;
}

_TEST test_Initializing_StartMoveAbsolute(void)
{
	PaddleMotorFB.PaddleMotor->STS.EndButtonHit = 1;
	PaddleMotorFB.PaddleMotor->STS.TimerEnded = 1;
	PaddleMotorFB.PaddleMotor->STS.ReferenceSet = 0;

	PaddleMotorFB.PaddleMotor->STS.ActPosition = 4000;

	FB_PaddleMotor(&PaddleMotorFB);

	TEST_ASSERT_EQUAL_INT(1, PaddleMotorFB.PaddleMotor->CS.MoveAbsolute);

	TEST_DONE;
}

_TEST test_Initializing_TargetPosition(void)
{
	PaddleMotorFB.PaddleMotor->STS.EndButtonHit = 1;
	PaddleMotorFB.PaddleMotor->STS.TimerEnded = 1;
	PaddleMotorFB.PaddleMotor->STS.ReferenceSet = 0;

	PaddleMotorFB.PaddleMotor->STS.ActPosition = 5000;

	FB_PaddleMotor(&PaddleMotorFB);

	TEST_ASSERT_EQUAL_INT(
		PaddleMotorFB.PaddleMotor->STS.ReferencePosition - MIDDLE_POSITION,
		PaddleMotorFB.PaddleMotor->PAR.Position
		);

	TEST_DONE;
}
/*
B+R UnitTest: This is generated code.
Do not edit! Do not move!
Description: UnitTest Testprogramm infrastructure (TestSet).
LastUpdated: 2026-05-01 11:41:13Z
By B+R UnitTest Helper Version: 2.0.2.35
*/
UNITTEST_FIXTURES(fixtures)
{
	new_TestFixture("test_Initializing_SetsParameters", test_Initializing_SetsParameters),
	new_TestFixture("test_Initializing_StartsHoming", test_Initializing_StartsHoming),
	new_TestFixture("test_Initializing_EndButtonHit", test_Initializing_EndButtonHit),
	new_TestFixture("test_Initializing_ToIdle", test_Initializing_ToIdle),
	new_TestFixture("test_Initializing_ReferencePosition", test_Initializing_ReferencePosition),
	new_TestFixture("test_Initializing_StartMoveAbsolute", test_Initializing_StartMoveAbsolute),
	new_TestFixture("test_Initializing_TargetPosition", test_Initializing_TargetPosition),
};

UNITTEST_CALLER_COMPLETE_EXPLICIT(testSet_PaddleMotor_Initializing, "testSet_PaddleMotor_Initializing", setupTest, 0, fixtures, 0, 0, 0);
```

#### testSet_PaddleMotor_Running.c
```c
/********************************************************************
 * COPYRIGHT - MyAutoMation-IT
 ********************************************************************
 * Author: Raivo Berends
 ********************************************************************/

#include <bur/plctypes.h>

#ifdef _DEFAULT_INCLUDES
#include <AsDefault.h>
#endif

#include "UnitTest.h"
#include "Library.h"
#include "CommonTypes.h"
#include <string.h>

_SETUP_TEST(void)
{
	PaddleMotorFB.PaddleMotor = &PaddleMotorStruct;

	// volledige reset van alles
	memset(PaddleMotorFB.PaddleMotor, 0, sizeof(*PaddleMotorFB.PaddleMotor));

	// minimale state voor RUNNING tests
	PaddleMotorFB.PaddleMotor->STS.StateInt = STATE_RUNNING;

	TEST_DONE;
}

_TEST test_Running_SetsFlagsCorrectly(void)
{
	PaddleMotorFB.PaddleMotor->STS.Idle = 1;

	FB_PaddleMotor(&PaddleMotorFB);

	TEST_ASSERT_EQUAL_INT(1, PaddleMotorFB.PaddleMotor->STS.Running);
	TEST_ASSERT_EQUAL_INT(0, PaddleMotorFB.PaddleMotor->STS.Idle);

	TEST_DONE;
}

_TEST test_Running_ManualMode_StopsJogging(void)
{
	PaddleMotorFB.PaddleMotor->CS.AutoMode = 0;

	PaddleMotorFB.PaddleMotor->CS.MoveJogNeg = 1;
	PaddleMotorFB.PaddleMotor->CS.MoveJogPos = 1;

	FB_PaddleMotor(&PaddleMotorFB);

	TEST_ASSERT_EQUAL_INT(0, PaddleMotorFB.PaddleMotor->CS.MoveJogNeg);
	TEST_ASSERT_EQUAL_INT(0, PaddleMotorFB.PaddleMotor->CS.MoveJogPos);

	TEST_DONE;
}

_TEST test_Running_IncreaseJogSpeed(void)
{
	PaddleMotorFB.PaddleMotor->CS.AutoMode = 0;

	PaddleMotorFB.PaddleMotor->PAR.JogVelocity = 500;
	PaddleMotorFB.PaddleMotor->HMI.IncreaseJogSpeed = 1;

	FB_PaddleMotor(&PaddleMotorFB);

	TEST_ASSERT_EQUAL_INT(501, PaddleMotorFB.PaddleMotor->PAR.JogVelocity);

	TEST_DONE;
}

_TEST test_Running_DecreaseJogSpeed(void)
{
	PaddleMotorFB.PaddleMotor->CS.AutoMode = 0;

	PaddleMotorFB.PaddleMotor->PAR.JogVelocity = 500;
	PaddleMotorFB.PaddleMotor->HMI.DecreaseJogSpeed = 1;

	FB_PaddleMotor(&PaddleMotorFB);

	TEST_ASSERT_EQUAL_INT(499, PaddleMotorFB.PaddleMotor->PAR.JogVelocity);

	TEST_DONE;
}

_TEST test_Running_IncreaseAccDec(void)
{
	PaddleMotorFB.PaddleMotor->CS.AutoMode = 0;

	PaddleMotorFB.PaddleMotor->PAR.Acceleration = 1000;
	PaddleMotorFB.PaddleMotor->PAR.Deceleration = 1000;

	PaddleMotorFB.PaddleMotor->HMI.IncreaseAccDec = 1;

	FB_PaddleMotor(&PaddleMotorFB);

	TEST_ASSERT_EQUAL_INT(1010, PaddleMotorFB.PaddleMotor->PAR.Acceleration);
	TEST_ASSERT_EQUAL_INT(1010, PaddleMotorFB.PaddleMotor->PAR.Deceleration);

	TEST_DONE;
}

_TEST test_Running_DecreaseAccDec(void)
{
	PaddleMotorFB.PaddleMotor->CS.AutoMode = 0;

	PaddleMotorFB.PaddleMotor->PAR.Acceleration = 2000;
	PaddleMotorFB.PaddleMotor->PAR.Deceleration = 2000;

	PaddleMotorFB.PaddleMotor->HMI.DecreaseAccDec = 1;

	FB_PaddleMotor(&PaddleMotorFB);

	TEST_ASSERT_EQUAL_INT(1990, PaddleMotorFB.PaddleMotor->PAR.Acceleration);
	TEST_ASSERT_EQUAL_INT(1990, PaddleMotorFB.PaddleMotor->PAR.Deceleration);

	TEST_DONE;
}

_TEST test_Running_AutoMode_ResetsHMIInputs(void)
{
	PaddleMotorFB.PaddleMotor->STS.AutoActive = 1;

	PaddleMotorFB.PaddleMotor->HMI.MoveJogNeg = 1;
	PaddleMotorFB.PaddleMotor->HMI.MoveJogPos = 1;
	PaddleMotorFB.PaddleMotor->HMI.MoveAbsolute = 1;

	FB_PaddleMotor(&PaddleMotorFB);

	TEST_ASSERT_EQUAL_INT(0, PaddleMotorFB.PaddleMotor->HMI.MoveJogNeg);
	TEST_ASSERT_EQUAL_INT(0, PaddleMotorFB.PaddleMotor->HMI.MoveJogPos);
	TEST_ASSERT_EQUAL_INT(0, PaddleMotorFB.PaddleMotor->HMI.MoveAbsolute);

	TEST_DONE;
}

_TEST test_Running_LowerLimitProtection(void)
{
	PaddleMotorFB.PaddleMotor->STS.ReferencePosition = 5000;
	PaddleMotorFB.PaddleMotor->STS.ActPosition = 1000;
	PaddleMotorFB.PaddleMotor->STS.ActVelocity = 0;

	FB_PaddleMotor(&PaddleMotorFB);

	TEST_ASSERT_EQUAL_INT(0, PaddleMotorFB.PaddleMotor->CS.MoveJogNeg);

	TEST_DONE;
}

_TEST test_Running_UpperLimitProtection_EndButton(void)
{
	PaddleMotorFB.digitalInput = 0x1;

	FB_PaddleMotor(&PaddleMotorFB);

	TEST_ASSERT_EQUAL_INT(0, PaddleMotorFB.PaddleMotor->CS.MoveJogPos);

	TEST_DONE;
}

_TEST test_Running_UpperLimitProtection_Position(void)
{
	PaddleMotorFB.PaddleMotor->STS.ReferencePosition = 5000;
	PaddleMotorFB.PaddleMotor->STS.ActPosition = 4900;
	PaddleMotorFB.PaddleMotor->STS.ActVelocity = 0;

	FB_PaddleMotor(&PaddleMotorFB);

	TEST_ASSERT_EQUAL_INT(0, PaddleMotorFB.PaddleMotor->CS.MoveJogPos);

	TEST_DONE;
}

_TEST test_Running_StoppingOffset_HighVelocityLimitsMovement(void)
{
	PaddleMotorFB.PaddleMotor->STS.ReferencePosition = 5000;

	// Hoge snelheid ? grote stopping offset
	PaddleMotorFB.PaddleMotor->STS.ActVelocity = 1000;

	// Dicht bij ondergrens
	PaddleMotorFB.PaddleMotor->STS.ActPosition = 2300;

	FB_PaddleMotor(&PaddleMotorFB);

	TEST_ASSERT_EQUAL_INT(0, PaddleMotorFB.PaddleMotor->CS.MoveJogNeg);

	TEST_DONE;
}

_TEST test_Running_LowerLimit_AdjustsTargetPosition(void)
{
	PaddleMotorFB.PaddleMotor->STS.ReferencePosition = 5000;
	PaddleMotorFB.PaddleMotor->STS.ActVelocity = 0;

	// Onder minimum grens
	PaddleMotorFB.PaddleMotor->STS.ActPosition = 1000;

	FB_PaddleMotor(&PaddleMotorFB);

	TEST_ASSERT_EQUAL_INT(PaddleMotorFB.PaddleMotor->STS.ActPosition + 100, PaddleMotorFB.PaddleMotor->PAR.Position);

	TEST_DONE;
}

_TEST test_Running_UpperLimit_AdjustsTargetPosition(void)
{
	PaddleMotorFB.PaddleMotor->STS.ReferencePosition = 5000;
	PaddleMotorFB.PaddleMotor->STS.ActVelocity = 0;

	// Dicht bij bovengrens
	PaddleMotorFB.PaddleMotor->STS.ActPosition = 4950;

	FB_PaddleMotor(&PaddleMotorFB);

	TEST_ASSERT_EQUAL_INT(PaddleMotorFB.PaddleMotor->STS.ReferencePosition - 100, PaddleMotorFB.PaddleMotor->PAR.Position);

	TEST_DONE;
}

_TEST test_Running_EndButton_ForcesStopJogPos(void)
{
	// Activeer endbutton
	PaddleMotorFB.digitalInput = 0x1;

	PaddleMotorFB.PaddleMotor->CS.MoveJogPos = 1;

	FB_PaddleMotor(&PaddleMotorFB);

	TEST_ASSERT_EQUAL_INT(0, PaddleMotorFB.PaddleMotor->CS.MoveJogPos);

	TEST_DONE;
}

_TEST test_Running_StopGame_TransitionsToStopping(void)
{
	PaddleMotorFB.PaddleMotor->CS.StopGame = 1;

	FB_PaddleMotor(&PaddleMotorFB);

	TEST_ASSERT_EQUAL_INT(STATE_STOPPING, PaddleMotorFB.PaddleMotor->STS.StateInt);

	TEST_DONE;
}

_TEST test_Running_StoppingOffset_AffectsUpperLimit(void)
{
	PaddleMotorFB.PaddleMotor->STS.ReferencePosition = 5000;

	// Zonder velocity ? geen offset
	PaddleMotorFB.PaddleMotor->STS.ActVelocity = 0;
	PaddleMotorFB.PaddleMotor->STS.ActPosition = 4900;

	FB_PaddleMotor(&PaddleMotorFB);

	int pos_no_offset = PaddleMotorFB.PaddleMotor->PAR.Position;

	// Reset situatie
	PaddleMotorFB.PaddleMotor->STS.ActVelocity = 1000;
	PaddleMotorFB.PaddleMotor->STS.ActPosition = 4900;

	FB_PaddleMotor(&PaddleMotorFB);

	int pos_with_offset = PaddleMotorFB.PaddleMotor->PAR.Position;

	TEST_ASSERT(pos_with_offset <= pos_no_offset);

	TEST_DONE;
}

/*
B+R UnitTest: This is generated code.
Do not edit! Do not move!
Description: UnitTest Testprogramm infrastructure (TestSet).
LastUpdated: 2026-05-01 12:04:37Z
By B+R UnitTest Helper Version: 2.0.2.35
*/
UNITTEST_FIXTURES(fixtures)
{
	new_TestFixture("test_Running_SetsFlagsCorrectly", test_Running_SetsFlagsCorrectly),
	new_TestFixture("test_Running_ManualMode_StopsJogging", test_Running_ManualMode_StopsJogging),
	new_TestFixture("test_Running_IncreaseJogSpeed", test_Running_IncreaseJogSpeed),
	new_TestFixture("test_Running_DecreaseJogSpeed", test_Running_DecreaseJogSpeed),
	new_TestFixture("test_Running_IncreaseAccDec", test_Running_IncreaseAccDec),
	new_TestFixture("test_Running_DecreaseAccDec", test_Running_DecreaseAccDec),
	new_TestFixture("test_Running_AutoMode_ResetsHMIInputs", test_Running_AutoMode_ResetsHMIInputs),
	new_TestFixture("test_Running_LowerLimitProtection", test_Running_LowerLimitProtection),
	new_TestFixture("test_Running_UpperLimitProtection_EndButton", test_Running_UpperLimitProtection_EndButton),
	new_TestFixture("test_Running_UpperLimitProtection_Position", test_Running_UpperLimitProtection_Position),
	new_TestFixture("test_Running_StoppingOffset_HighVelocityLimitsMovement", test_Running_StoppingOffset_HighVelocityLimitsMovement),
	new_TestFixture("test_Running_LowerLimit_AdjustsTargetPosition", test_Running_LowerLimit_AdjustsTargetPosition),
	new_TestFixture("test_Running_UpperLimit_AdjustsTargetPosition", test_Running_UpperLimit_AdjustsTargetPosition),
	new_TestFixture("test_Running_EndButton_ForcesStopJogPos", test_Running_EndButton_ForcesStopJogPos),
	new_TestFixture("test_Running_StopGame_TransitionsToStopping", test_Running_StopGame_TransitionsToStopping),
	new_TestFixture("test_Running_StoppingOffset_AffectsUpperLimit", test_Running_StoppingOffset_AffectsUpperLimit),
};

UNITTEST_CALLER_COMPLETE_EXPLICIT(testSet_PaddleMotor_Running, "testSet_PaddleMotor_Running", setupTest, 0, fixtures, 0, 0, 0);
```

#### testSet_PaddleMotor_Stopping.c
```c
/********************************************************************
 * COPYRIGHT - MyAutoMation-IT
 ********************************************************************
 * Author: Raivo Berends
 ********************************************************************/

#include <bur/plctypes.h>

#ifdef _DEFAULT_INCLUDES
#include <AsDefault.h>
#endif

#include "UnitTest.h"
#include "Library.h"
#include "CommonTypes.h"
#include <string.h>

_SETUP_TEST(void)
{
	PaddleMotorFB.PaddleMotor = &PaddleMotorStruct;
	memset(PaddleMotorFB.PaddleMotor, 0, sizeof(*PaddleMotorFB.PaddleMotor));
	PaddleMotorFB.PaddleMotor->STS.StateInt = STATE_STOPPING;

	TEST_DONE;
}

_TEST test_Stopping_AllCommandsReset(void)
{
	FB_PaddleMotor(&PaddleMotorFB);

	TEST_ASSERT_EQUAL_INT(0, PaddleMotorFB.PaddleMotor->CS.MoveAbsolute);
	TEST_ASSERT_EQUAL_INT(0, PaddleMotorFB.PaddleMotor->CS.MoveJogNeg);
	TEST_ASSERT_EQUAL_INT(0, PaddleMotorFB.PaddleMotor->CS.MoveJogPos);
	TEST_ASSERT_EQUAL_INT(1, PaddleMotorFB.PaddleMotor->CS.Stop);

	TEST_DONE;
}

_TEST test_Stopping_RemainsInState_WhenNotStandStill(void)
{
	PaddleMotorFB.PaddleMotor->STS.StandStill = 0;
	PaddleMotorFB.PaddleMotor->STS.Interlocked = 0;

	FB_PaddleMotor(&PaddleMotorFB);

	TEST_ASSERT_EQUAL_INT(STATE_STOPPING, PaddleMotorFB.PaddleMotor->STS.StateInt);

	TEST_DONE;
}

_TEST test_Stopping_ToDisabled_WhenStandStill(void)
{
	PaddleMotorFB.PaddleMotor->STS.StandStill = 1;
	PaddleMotorFB.PaddleMotor->STS.Interlocked = 0;

	FB_PaddleMotor(&PaddleMotorFB);

	TEST_ASSERT_EQUAL_INT(STATE_DISABLED, PaddleMotorFB.PaddleMotor->STS.StateInt);

	TEST_DONE;
}

_TEST test_Stopping_NoTransition_WhenInterlocked(void)
{
	PaddleMotorFB.PaddleMotor->STS.StandStill = 1;
	PaddleMotorFB.PaddleMotor->STS.Interlocked = 1;

	FB_PaddleMotor(&PaddleMotorFB);

	TEST_ASSERT_EQUAL_INT(STATE_STOPPING, PaddleMotorFB.PaddleMotor->STS.StateInt);

	TEST_DONE;
}

_TEST test_Stopping_StopSignalAlwaysActive(void)
{
	FB_PaddleMotor(&PaddleMotorFB);

	TEST_ASSERT_EQUAL_INT(1, PaddleMotorFB.PaddleMotor->CS.Stop);

	TEST_DONE;
}

/*
B+R UnitTest: This is generated code.
Do not edit! Do not move!
Description: UnitTest Testprogramm infrastructure (TestSet).
LastUpdated: 2026-05-01 12:04:37Z
By B+R UnitTest Helper Version: 2.0.2.35
*/
UNITTEST_FIXTURES(fixtures)
{
	new_TestFixture("test_Stopping_AllCommandsReset", test_Stopping_AllCommandsReset),
	new_TestFixture("test_Stopping_RemainsInState_WhenNotStandStill", test_Stopping_RemainsInState_WhenNotStandStill),
	new_TestFixture("test_Stopping_ToDisabled_WhenStandStill", test_Stopping_ToDisabled_WhenStandStill),
	new_TestFixture("test_Stopping_NoTransition_WhenInterlocked", test_Stopping_NoTransition_WhenInterlocked),
	new_TestFixture("test_Stopping_StopSignalAlwaysActive", test_Stopping_StopSignalAlwaysActive),
};

UNITTEST_CALLER_COMPLETE_EXPLICIT(testSet_PaddleMotor_Stopping, "testSet_PaddleMotor_Stopping", setupTest, 0, fixtures, 0, 0, 0);
```

#### testSuite.c
```c
/********************************************************************
 * COPYRIGHT --
 ********************************************************************
 * Program: -
 * Author:
 * Created:
 ********************************************************************
 * Test registration and handshake
 ********************************************************************/

#include <bur/plctypes.h>

#ifdef _DEFAULT_INCLUDES
#include <AsDefault.h>
#endif

#include "UnitTest.h"
#include "Library.h"

void _INIT initTestSuite(void)
{
	utInit(&Testsuite);
}

void _CYCLIC cyclicWithTest(void)
{
	utCyclic(&Testsuite);
}

void _EXIT exitTestSuite(void)
{
	utExit(&Testsuite);
}
```

### Package Logical/UnitTests/UnitTests/TestSet_Templates - Multiple variants of valid test sets

### testSet_Template.c
```c
/********************************************************************
 * COPYRIGHT - MyAutoMation-IT
 ********************************************************************
 * Author: Raivo Berends
 ********************************************************************/

#include <bur/plctypes.h>

#ifdef _DEFAULT_INCLUDES
#include <AsDefault.h>
#endif

#include "UnitTest.h"
#include "Library.h"
#include "CommonTypes.h"

_SETUP_TEST(void)
{
	PaddleMotorFB.PaddleMotor = &PaddleMotorStruct;
	PaddleMotorFB.PaddleMotor->STS.StateInt = STATE_IDLE;

	TEST_DONE;
}

_TEST test_Template(void)
{
}

/*
B+R UnitTest: This is generated code.
Do not edit! Do not move!
Description: UnitTest Testprogramm infrastructure (TestSet).
LastUpdated: 2026-05-01 11:23:13Z
By B+R UnitTest Helper Version: 2.0.2.35
*/
UNITTEST_FIXTURES(fixtures)
{
};

UNITTEST_CALLER_COMPLETE_EXPLICIT(testSet_PaddleMotor_Idle, "testSet_Template", setupTest, 0, fixtures, 0, 0, 0);
```

### Program Logical/UnitTests/UnitTests/Tests_BallControl_C (ANSIC)

#### variables.var - Name the suite and add PVs for the program
```iecst
(********************************************************************
 * COPYRIGHT --  MyAutomation-IT
 ********************************************************************
 * Program: Tests_BallControl_C
 * File: variables.var
 * Author: Raivo Berends
 ********************************************************************
 * Local variables of program Tests_BallControl_C
 ********************************************************************)
(*Describe the test*)
VAR
	Testsuite : UtMgrTestSuite := (Name:='BallControl_Tests',Type:=utMgrTEST_TYPE_C);
END_VAR
(*Variables used in the tests*)
VAR
	BallControlFB : FB_BallControl;
	DistanceSensorLeftStruct : UDT_DistanceSensor;
	DistanceSensorMiddleStruct : UDT_DistanceSensor;
	DistanceSensorRightStruct : UDT_DistanceSensor;
	BallControlStruct : UDT_BallControl;
	PaddleMotorStruct : UDT_PaddleMotor;
	ShooterStruct : UDT_Shooter;
END_VAR
```

#### autoGeneratedFile.c - Auto generated code - list of all test sets in the program
```c
/*
B+R UnitTest: This is generated code.
Do not edit! Do not move!
Description: UnitTest Testprogramm infrastructure (List of TestSets).
LastUpdated: 2026-05-07 12:26:03Z
By B+R UnitTest Helper Version: 2.0.2.35
*/
#include "UnitTest.h"

UNITTEST_TESTSET_DECLARATION  testSet_BallControl_Disabled;
UNITTEST_TESTSET_DECLARATION  testSet_BallControl_Initializing;
UNITTEST_TESTSET_DECLARATION  testSet_BallControl_Idle;
UNITTEST_TESTSET_DECLARATION  testSet_BallControl_Running;
UNITTEST_TESTSET_DECLARATION  testSet_BallControl_Stopping;

UNITTEST_TESTSET_FIXTURES(utTestSets)
{
	new_TestSet(testSet_BallControl_Disabled),
	new_TestSet(testSet_BallControl_Initializing),
	new_TestSet(testSet_BallControl_Idle),
	new_TestSet(testSet_BallControl_Running),
	new_TestSet(testSet_BallControl_Stopping),
};
UNTITTEST_TESTSET_HANDLER();
```

#### testSet_BallControl_Disabled.c
```c
/********************************************************************
 * COPYRIGHT - MyAutoMation-IT
 ********************************************************************
 * Author: Raivo Berends
 ********************************************************************/

#include <bur/plctypes.h>

#ifdef _DEFAULT_INCLUDES
#include <AsDefault.h>
#endif

#include "UnitTest.h"
#include "Library.h"
#include "CommonTypes.h"
#include <string.h>

_SETUP_TEST(void)
{
	BallControlFB.BallControl = &BallControlStruct;
	BallControlFB.DistanceSensorLeft = &DistanceSensorLeftStruct;
	BallControlFB.DistanceSensorMiddle = &DistanceSensorMiddleStruct;
	BallControlFB.DistanceSensorRight = &DistanceSensorRightStruct;
	BallControlFB.PaddleMotor = &PaddleMotorStruct;
	BallControlFB.Shooter = &ShooterStruct;

	memset(BallControlFB.BallControl, 0, sizeof(*BallControlFB.BallControl));
	memset(BallControlFB.DistanceSensorLeft, 0, sizeof(*BallControlFB.DistanceSensorLeft));
	memset(BallControlFB.DistanceSensorMiddle, 0, sizeof(*BallControlFB.DistanceSensorMiddle));
	memset(BallControlFB.DistanceSensorRight, 0, sizeof(*BallControlFB.DistanceSensorRight));
	memset(BallControlFB.PaddleMotor, 0, sizeof(*BallControlFB.PaddleMotor));
	memset(BallControlFB.Shooter, 0, sizeof(*BallControlFB.Shooter));

	BallControlFB.BallControl->STS.StateInt = STATE_DISABLED;

	TEST_DONE;
}

_TEST Test_Disabled_ResetsShoot(void)
{
	BallControlFB.BallControl->CS.Shoot = 1;

	FB_BallControl(&BallControlFB);

	TEST_ASSERT_EQUAL_INT(0, BallControlFB.BallControl->CS.Shoot);

	TEST_DONE;
}

_TEST Test_Disabled_IntensityIncrease(void)
{
	BallControlFB.Shooter->HMI.IncreaseIntensity = 1;
	BallControlFB.Shooter->PAR.Intensity = 5;

	FB_BallControl(&BallControlFB);

	TEST_ASSERT(BallControlFB.Shooter->PAR.Intensity > 5);

	TEST_DONE;
}

_TEST Test_Disabled_IntensityDecrease(void)
{
	BallControlFB.Shooter->HMI.DecreaseIntensity = 1;
	BallControlFB.Shooter->PAR.Intensity = 5;

	FB_BallControl(&BallControlFB);

	TEST_ASSERT(BallControlFB.Shooter->PAR.Intensity < 5);

	TEST_DONE;
}

_TEST Test_Disabled_IntensityUpperLimit(void)
{
	BallControlFB.Shooter->HMI.IncreaseIntensity = 1;
	BallControlFB.Shooter->PAR.Intensity = MAX_INTENSITY;

	FB_BallControl(&BallControlFB);

	TEST_ASSERT_EQUAL_INT(MAX_INTENSITY, BallControlFB.Shooter->PAR.Intensity);

	TEST_DONE;
}

_TEST Test_Disabled_IntensityLowerLimit(void)
{
	BallControlFB.Shooter->HMI.DecreaseIntensity = 1;
	BallControlFB.Shooter->PAR.Intensity = MIN_INTENSITY;

	FB_BallControl(&BallControlFB);

	TEST_ASSERT_EQUAL_INT(MIN_INTENSITY, BallControlFB.Shooter->PAR.Intensity);

	TEST_DONE;
}

_TEST Test_Disabled_TransitionsToInitializing(void)
{
	BallControlFB.BallControl->STS.Initializing = 1;

	FB_BallControl(&BallControlFB);

	TEST_ASSERT_EQUAL_INT(STATE_INITIALIZING, BallControlFB.BallControl->STS.StateInt);

	TEST_DONE;
}

_TEST Test_Disabled_NoTransitionWithoutInit(void)
{
	BallControlFB.BallControl->STS.Initializing = 0;

	FB_BallControl(&BallControlFB);

	TEST_ASSERT_EQUAL_INT(STATE_DISABLED, BallControlFB.BallControl->STS.StateInt);

	TEST_DONE;
}

_TEST Test_Disabled_StopsOnlyShootCommand(void)
{
	BallControlFB.BallControl->CS.Shoot = 1;
	BallControlFB.BallControl->CS.AutoMode = 1;

	FB_BallControl(&BallControlFB);

	TEST_ASSERT_EQUAL_INT(0, BallControlFB.BallControl->CS.Shoot);
	TEST_ASSERT_EQUAL_INT(1, BallControlFB.BallControl->CS.AutoMode);

	TEST_DONE;
}

/*
B+R UnitTest: This is generated code.
Do not edit! Do not move!
Description: UnitTest Testprogramm infrastructure (TestSet).
LastUpdated: 2026-05-07 11:56:27Z
By B+R UnitTest Helper Version: 2.0.2.35
*/
UNITTEST_FIXTURES(fixtures)
{
	new_TestFixture("Test_Disabled_ResetsShoot", Test_Disabled_ResetsShoot),
	new_TestFixture("Test_Disabled_IntensityIncrease", Test_Disabled_IntensityIncrease),
	new_TestFixture("Test_Disabled_IntensityDecrease", Test_Disabled_IntensityDecrease),
	new_TestFixture("Test_Disabled_IntensityUpperLimit", Test_Disabled_IntensityUpperLimit),
	new_TestFixture("Test_Disabled_IntensityLowerLimit", Test_Disabled_IntensityLowerLimit),
	new_TestFixture("Test_Disabled_TransitionsToInitializing", Test_Disabled_TransitionsToInitializing),
	new_TestFixture("Test_Disabled_NoTransitionWithoutInit", Test_Disabled_NoTransitionWithoutInit),
	new_TestFixture("Test_Disabled_StopsOnlyShootCommand", Test_Disabled_StopsOnlyShootCommand),
};

UNITTEST_CALLER_COMPLETE_EXPLICIT(testSet_BallControl_Disabled, "testSet_BallControl_Disabled", setupTest, 0, fixtures, 0, 0, 0);
```

#### testSet_BallControl_Initializing.c
```c
/********************************************************************
 * COPYRIGHT - MyAutoMation-IT
 ********************************************************************
 * Author: Raivo Berends
 ********************************************************************/

#include <bur/plctypes.h>

#ifdef _DEFAULT_INCLUDES
#include <AsDefault.h>
#endif

#include "UnitTest.h"
#include "Library.h"
#include "CommonTypes.h"
#include <string.h>

_SETUP_TEST(void)
{
	BallControlFB.BallControl = &BallControlStruct;
	BallControlFB.DistanceSensorLeft = &DistanceSensorLeftStruct;
	BallControlFB.DistanceSensorMiddle = &DistanceSensorMiddleStruct;
	BallControlFB.DistanceSensorRight = &DistanceSensorRightStruct;
	BallControlFB.PaddleMotor = &PaddleMotorStruct;
	BallControlFB.Shooter = &ShooterStruct;

	memset(BallControlFB.BallControl, 0, sizeof(*BallControlFB.BallControl));
	memset(BallControlFB.DistanceSensorLeft, 0, sizeof(*BallControlFB.DistanceSensorLeft));
	memset(BallControlFB.DistanceSensorMiddle, 0, sizeof(*BallControlFB.DistanceSensorMiddle));
	memset(BallControlFB.DistanceSensorRight, 0, sizeof(*BallControlFB.DistanceSensorRight));
	memset(BallControlFB.PaddleMotor, 0, sizeof(*BallControlFB.PaddleMotor));
	memset(BallControlFB.Shooter, 0, sizeof(*BallControlFB.Shooter));

	BallControlFB.BallControl->STS.StateInt = STATE_INITIALIZING;

	TEST_DONE;
}

_TEST Test_Initializing_ResetsStates(void)
{
	BallControlFB.BallControl->STS.PrevShootState = 5;
	BallControlFB.BallControl->STS.ShootState = 10;
	BallControlFB.BallControl->STS.GameOver = 1;
	BallControlFB.BallControl->STS.FirstRun = 0;

	FB_BallControl(&BallControlFB);

	TEST_ASSERT_EQUAL_INT(0, BallControlFB.BallControl->STS.PrevShootState);
	TEST_ASSERT_EQUAL_INT(0, BallControlFB.BallControl->STS.ShootState);
	TEST_ASSERT_EQUAL_INT(0, BallControlFB.BallControl->STS.GameOver);
	TEST_ASSERT_EQUAL_INT(1, BallControlFB.BallControl->STS.FirstRun);

	TEST_DONE;
}

_TEST Test_Initializing_TransitionsToIdle(void)
{
	BallControlFB.BallControl->STS.Idle = 1;

	FB_BallControl(&BallControlFB);

	TEST_ASSERT_EQUAL_INT(STATE_IDLE, BallControlFB.BallControl->STS.StateInt);

	TEST_DONE;
}

_TEST Test_Initializing_NoIdleStaysInState(void)
{;
	BallControlFB.BallControl->STS.Idle = 0;

	FB_BallControl(&BallControlFB);

	TEST_ASSERT_EQUAL_INT(STATE_INITIALIZING, BallControlFB.BallControl->STS.StateInt);

	TEST_DONE;
}

/*
B+R UnitTest: This is generated code.
Do not edit! Do not move!
Description: UnitTest Testprogramm infrastructure (TestSet).
LastUpdated: 2026-05-07 12:20:57Z
By B+R UnitTest Helper Version: 2.0.2.35
*/
UNITTEST_FIXTURES(fixtures)
{
	new_TestFixture("Test_Initializing_ResetsStates", Test_Initializing_ResetsStates),
	new_TestFixture("Test_Initializing_TransitionsToIdle", Test_Initializing_TransitionsToIdle),
	new_TestFixture("Test_Initializing_NoIdleStaysInState", Test_Initializing_NoIdleStaysInState),
};

UNITTEST_CALLER_COMPLETE_EXPLICIT(testSet_BallControl_Initializing, "testSet_BallControl_Initializing", setupTest, 0, fixtures, 0, 0, 0);
```

#### testSet_BallControl_Idle.c
```c
/********************************************************************
 * COPYRIGHT - MyAutoMation-IT
 ********************************************************************
 * Author: Raivo Berends
 ********************************************************************/

#include <bur/plctypes.h>

#ifdef _DEFAULT_INCLUDES
#include <AsDefault.h>
#endif

#include "UnitTest.h"
#include "Library.h"
#include "CommonTypes.h"
#include <string.h>

_SETUP_TEST(void)
{
	BallControlFB.BallControl = &BallControlStruct;
	BallControlFB.DistanceSensorLeft = &DistanceSensorLeftStruct;
	BallControlFB.DistanceSensorMiddle = &DistanceSensorMiddleStruct;
	BallControlFB.DistanceSensorRight = &DistanceSensorRightStruct;
	BallControlFB.PaddleMotor = &PaddleMotorStruct;
	BallControlFB.Shooter = &ShooterStruct;

	memset(BallControlFB.BallControl, 0, sizeof(*BallControlFB.BallControl));
	memset(BallControlFB.DistanceSensorLeft, 0, sizeof(*BallControlFB.DistanceSensorLeft));
	memset(BallControlFB.DistanceSensorMiddle, 0, sizeof(*BallControlFB.DistanceSensorMiddle));
	memset(BallControlFB.DistanceSensorRight, 0, sizeof(*BallControlFB.DistanceSensorRight));
	memset(BallControlFB.PaddleMotor, 0, sizeof(*BallControlFB.PaddleMotor));
	memset(BallControlFB.Shooter, 0, sizeof(*BallControlFB.Shooter));

	BallControlFB.BallControl->STS.StateInt = STATE_IDLE;

	TEST_DONE;
}

_TEST Test_Idle_StaysIdle_WhenNotRunning(void)
{
	BallControlFB.BallControl->STS.Running = 0;

	FB_BallControl(&BallControlFB);

	TEST_ASSERT_EQUAL_INT(STATE_IDLE, BallControlFB.BallControl->STS.StateInt);

	TEST_DONE;
}

_TEST Test_Idle_TransitionsToRunning_WhenRunningTrue(void)
{
	BallControlFB.BallControl->STS.Running = 1;

	FB_BallControl(&BallControlFB);

	TEST_ASSERT_EQUAL_INT(STATE_RUNNING, BallControlFB.BallControl->STS.StateInt);

	TEST_DONE;
}

_TEST Test_Idle_TransitionsOnlyOnRunningTrue(void)
{
	/* cycle 1: not running */
	BallControlFB.BallControl->STS.Running = 0;
	FB_BallControl(&BallControlFB);
	TEST_ASSERT_EQUAL_INT(STATE_IDLE, BallControlFB.BallControl->STS.StateInt);

	/* cycle 2: running becomes true */
	BallControlFB.BallControl->STS.Running = 1;
	FB_BallControl(&BallControlFB);
	TEST_ASSERT_EQUAL_INT(STATE_RUNNING, BallControlFB.BallControl->STS.StateInt);

	TEST_DONE;
}

/*
B+R UnitTest: This is generated code.
Do not edit! Do not move!
Description: UnitTest Testprogramm infrastructure (TestSet).
LastUpdated: 2026-05-07 12:26:03Z
By B+R UnitTest Helper Version: 2.0.2.35
*/
UNITTEST_FIXTURES(fixtures)
{
	new_TestFixture("Test_Idle_StaysIdle_WhenNotRunning", Test_Idle_StaysIdle_WhenNotRunning),
	new_TestFixture("Test_Idle_TransitionsToRunning_WhenRunningTrue", Test_Idle_TransitionsToRunning_WhenRunningTrue),
	new_TestFixture("Test_Idle_TransitionsOnlyOnRunningTrue", Test_Idle_TransitionsOnlyOnRunningTrue),
};

UNITTEST_CALLER_COMPLETE_EXPLICIT(testSet_BallControl_Idle, "testSet_BallControl_Idle", setupTest, 0, fixtures, 0, 0, 0);
```

#### testSet_BallControl_Running.c
```c
/********************************************************************
 * COPYRIGHT - MyAutoMation-IT
 ********************************************************************
 * Author: Raivo Berends
 ********************************************************************/

#include <bur/plctypes.h>

#ifdef _DEFAULT_INCLUDES
#include <AsDefault.h>
#endif

#include "UnitTest.h"
#include "Library.h"
#include "CommonTypes.h"
#include <string.h>

_SETUP_TEST(void)
{
	BallControlFB.BallControl = &BallControlStruct;
	BallControlFB.DistanceSensorLeft = &DistanceSensorLeftStruct;
	BallControlFB.DistanceSensorMiddle = &DistanceSensorMiddleStruct;
	BallControlFB.DistanceSensorRight = &DistanceSensorRightStruct;
	BallControlFB.PaddleMotor = &PaddleMotorStruct;
	BallControlFB.Shooter = &ShooterStruct;

	memset(BallControlFB.BallControl, 0, sizeof(*BallControlFB.BallControl));
	memset(BallControlFB.DistanceSensorLeft, 0, sizeof(*BallControlFB.DistanceSensorLeft));
	memset(BallControlFB.DistanceSensorMiddle, 0, sizeof(*BallControlFB.DistanceSensorMiddle));
	memset(BallControlFB.DistanceSensorRight, 0, sizeof(*BallControlFB.DistanceSensorRight));
	memset(BallControlFB.PaddleMotor, 0, sizeof(*BallControlFB.PaddleMotor));
	memset(BallControlFB.Shooter, 0, sizeof(*BallControlFB.Shooter));

	BallControlFB.BallControl->STS.StateInt = STATE_RUNNING;

	TEST_DONE;
}

_TEST Test_Running_AutoActive_SetsOutputs(void)
{
	BallControlFB.BallControl->STS.AutoActive = 1;

	FB_BallControl(&BallControlFB);

	TEST_ASSERT_EQUAL_INT(0, BallControlFB.PaddleMotor->CS.MoveAbsolute);
	TEST_ASSERT_EQUAL_INT(1, BallControlFB.Shooter->CS.EnableFan);
	TEST_ASSERT_EQUAL_INT(AUTOMODE_VELOCITY, BallControlFB.PaddleMotor->PAR.Velocity);

	TEST_DONE;
}

_TEST Test_Running_WhenAutoInactive_DisablesShoot(void)
{
	BallControlFB.BallControl->STS.AutoActive = 0;

	BallControlFB.BallControl->CS.Shoot = 1;

	FB_BallControl(&BallControlFB);

	TEST_ASSERT_EQUAL_INT(0, BallControlFB.BallControl->CS.Shoot);

	TEST_DONE;
}

_TEST Test_Running_State0_RightSensor_GoesToState5(void)
{
	BallControlFB.BallControl->STS.AutoActive = 1;

	BallControlFB.BallControl->STS.ShootState = 0;
	BallControlFB.BallControl->STS.FirstRun = 1;

	BallControlFB.DistanceSensorRight->STS.BallDetected = 1;

	FB_BallControl(&BallControlFB);

	TEST_ASSERT_EQUAL_INT(5, BallControlFB.BallControl->STS.ShootState);
	TEST_ASSERT_EQUAL_INT(0, BallControlFB.BallControl->STS.FirstRun);

	TEST_DONE;
}

_TEST Test_Running_State10_MiddleSensor_GoesToState20(void)
{
	BallControlFB.BallControl->STS.AutoActive = 1;

	BallControlFB.BallControl->STS.ShootState = 10;
	BallControlFB.DistanceSensorMiddle->STS.BallDetected = 1;

	FB_BallControl(&BallControlFB);

	TEST_ASSERT_EQUAL_INT(20, BallControlFB.BallControl->STS.ShootState);

	TEST_DONE;
}

_TEST Test_Running_State20_LeftSensor_GoesToState30(void)
{
	BallControlFB.BallControl->STS.AutoActive = 1;

	BallControlFB.BallControl->STS.ShootState = 20;
	BallControlFB.DistanceSensorLeft->STS.BallDetected = 1;

	FB_BallControl(&BallControlFB);

	TEST_ASSERT_EQUAL_INT(30, BallControlFB.BallControl->STS.ShootState);

	TEST_DONE;
}

_TEST Test_Running_State30_FiresShootAndResets(void)
{
	BallControlFB.BallControl->STS.AutoActive = 1;

	BallControlFB.BallControl->STS.ShootState = 30;

	FB_BallControl(&BallControlFB);

	TEST_ASSERT_EQUAL_INT(1, BallControlFB.BallControl->CS.Shoot);
	TEST_ASSERT_EQUAL_INT(0, BallControlFB.BallControl->STS.ShootState);

	TEST_DONE;
}

_TEST Test_Running_FirstRun_OnlyResetsOnce(void)
{
	BallControlFB.BallControl->STS.AutoActive = 1;

	BallControlFB.BallControl->STS.ShootState = 0;
	BallControlFB.BallControl->STS.FirstRun = 1;

	BallControlFB.DistanceSensorRight->STS.BallDetected = 1;

	FB_BallControl(&BallControlFB);

	TEST_ASSERT_EQUAL_INT(0, BallControlFB.BallControl->STS.FirstRun);

	TEST_DONE;
}

_TEST Test_Running_State0_NoBallDetected_StaysInState0(void)
{
	BallControlFB.BallControl->STS.AutoActive = 1;

	BallControlFB.BallControl->STS.ShootState = 0;
	BallControlFB.BallControl->STS.FirstRun = 1;

	BallControlFB.DistanceSensorRight->STS.BallDetected = 0;

	FB_BallControl(&BallControlFB);

	TEST_ASSERT_EQUAL_INT(0, BallControlFB.BallControl->STS.ShootState);
	TEST_ASSERT_EQUAL_INT(1, BallControlFB.BallControl->STS.FirstRun);

	TEST_DONE;
}

_TEST Test_Running_State10_NoMiddleDetection_StaysInState10(void)
{
	BallControlFB.BallControl->STS.AutoActive = 1;

	BallControlFB.BallControl->STS.ShootState = 10;

	BallControlFB.DistanceSensorMiddle->STS.BallDetected = 0;

	FB_BallControl(&BallControlFB);

	TEST_ASSERT_EQUAL_INT(10, BallControlFB.BallControl->STS.ShootState);

	TEST_DONE;
}

_TEST Test_Running_State20_NoLeftDetection_StaysInState20(void)
{
	BallControlFB.BallControl->STS.AutoActive = 1;

	BallControlFB.BallControl->STS.ShootState = 20;

	BallControlFB.DistanceSensorLeft->STS.BallDetected = 0;

	FB_BallControl(&BallControlFB);

	TEST_ASSERT_EQUAL_INT(20, BallControlFB.BallControl->STS.ShootState);

	TEST_DONE;
}

_TEST Test_Running_State0_FirstRunFalse_DoesNotTriggerState5(void)
{
	BallControlFB.BallControl->STS.AutoActive = 1;

	BallControlFB.BallControl->STS.FirstRun = 0;
	BallControlFB.BallControl->STS.ShootState = 0;

	BallControlFB.DistanceSensorRight->STS.BallDetected = 1;

	FB_BallControl(&BallControlFB);

	TEST_ASSERT_EQUAL_INT(0, BallControlFB.BallControl->STS.ShootState);

	TEST_DONE;
}

_TEST Test_Running_AutoInactive_DoesNotChangeShootState(void)
{
	BallControlFB.BallControl->STS.AutoActive = 0;

	BallControlFB.BallControl->STS.ShootState = 20;

	FB_BallControl(&BallControlFB);

	TEST_ASSERT_EQUAL_INT(20, BallControlFB.BallControl->STS.ShootState);

	TEST_DONE;
}

_TEST Test_Running_StopGame_TransitionsToStopping(void)
{
	BallControlFB.BallControl->CS.StopGame = 1;

	BallControlFB.BallControl->STS.AlarmActive = 0;
	BallControlFB.BallControl->STS.Interlocked = 0;

	FB_BallControl(&BallControlFB);

	TEST_ASSERT_EQUAL_INT(STATE_STOPPING, BallControlFB.BallControl->STS.StateInt);

	TEST_DONE;
}

_TEST Test_Running_StopGame_WithInterlock_DoesNotStop(void)
{
	BallControlFB.BallControl->CS.StopGame = 1;

	BallControlFB.BallControl->STS.AlarmActive = 0;
	BallControlFB.BallControl->STS.Interlocked = 1;

	FB_BallControl(&BallControlFB);

	TEST_ASSERT_EQUAL_INT(STATE_RUNNING, BallControlFB.BallControl->STS.StateInt);

	TEST_DONE;
}
/*
B+R UnitTest: This is generated code.
Do not edit! Do not move!
Description: UnitTest Testprogramm infrastructure (TestSet).
LastUpdated: 2026-05-08 07:54:53Z
By B+R UnitTest Helper Version: 2.0.2.35
*/
UNITTEST_FIXTURES(fixtures)
{
	new_TestFixture("Test_Running_AutoActive_SetsOutputs", Test_Running_AutoActive_SetsOutputs),
	new_TestFixture("Test_Running_WhenAutoInactive_DisablesShoot", Test_Running_WhenAutoInactive_DisablesShoot),
	new_TestFixture("Test_Running_State0_RightSensor_GoesToState5", Test_Running_State0_RightSensor_GoesToState5),
	new_TestFixture("Test_Running_State10_MiddleSensor_GoesToState20", Test_Running_State10_MiddleSensor_GoesToState20),
	new_TestFixture("Test_Running_State20_LeftSensor_GoesToState30", Test_Running_State20_LeftSensor_GoesToState30),
	new_TestFixture("Test_Running_State30_FiresShootAndResets", Test_Running_State30_FiresShootAndResets),
	new_TestFixture("Test_Running_FirstRun_OnlyResetsOnce", Test_Running_FirstRun_OnlyResetsOnce),
	new_TestFixture("Test_Running_State0_NoBallDetected_StaysInState0", Test_Running_State0_NoBallDetected_StaysInState0),
	new_TestFixture("Test_Running_State10_NoMiddleDetection_StaysInState10", Test_Running_State10_NoMiddleDetection_StaysInState10),
	new_TestFixture("Test_Running_State20_NoLeftDetection_StaysInState20", Test_Running_State20_NoLeftDetection_StaysInState20),
	new_TestFixture("Test_Running_State0_FirstRunFalse_DoesNotTriggerState5", Test_Running_State0_FirstRunFalse_DoesNotTriggerState5),
	new_TestFixture("Test_Running_AutoInactive_DoesNotChangeShootState", Test_Running_AutoInactive_DoesNotChangeShootState),
	new_TestFixture("Test_Running_StopGame_TransitionsToStopping", Test_Running_StopGame_TransitionsToStopping),
	new_TestFixture("Test_Running_StopGame_WithInterlock_DoesNotStop", Test_Running_StopGame_WithInterlock_DoesNotStop),
};

UNITTEST_CALLER_COMPLETE_EXPLICIT(testSet_BallControl_Running, "testSet_BallControl_Running", setupTest, 0, fixtures, 0, 0, 0);
```

#### testSet_BallControl_Stopping.c
```c
/********************************************************************
 * COPYRIGHT - MyAutoMation-IT
 ********************************************************************
 * Author: Raivo Berends
 ********************************************************************/

#include <bur/plctypes.h>

#ifdef _DEFAULT_INCLUDES
#include <AsDefault.h>
#endif

#include "UnitTest.h"
#include "Library.h"
#include "CommonTypes.h"
#include <string.h>

_SETUP_TEST(void)
{
	BallControlFB.BallControl = &BallControlStruct;
	BallControlFB.DistanceSensorLeft = &DistanceSensorLeftStruct;
	BallControlFB.DistanceSensorMiddle = &DistanceSensorMiddleStruct;
	BallControlFB.DistanceSensorRight = &DistanceSensorRightStruct;
	BallControlFB.PaddleMotor = &PaddleMotorStruct;
	BallControlFB.Shooter = &ShooterStruct;

	memset(BallControlFB.BallControl, 0, sizeof(*BallControlFB.BallControl));
	memset(BallControlFB.DistanceSensorLeft, 0, sizeof(*BallControlFB.DistanceSensorLeft));
	memset(BallControlFB.DistanceSensorMiddle, 0, sizeof(*BallControlFB.DistanceSensorMiddle));
	memset(BallControlFB.DistanceSensorRight, 0, sizeof(*BallControlFB.DistanceSensorRight));
	memset(BallControlFB.PaddleMotor, 0, sizeof(*BallControlFB.PaddleMotor));
	memset(BallControlFB.Shooter, 0, sizeof(*BallControlFB.Shooter));

	BallControlFB.BallControl->STS.StateInt = STATE_STOPPING;

	TEST_DONE;
}

_TEST Test_Stopping_StaysInStopping_WhenNotDisabled(void)
{
	BallControlFB.BallControl->STS.StateInt = STATE_STOPPING;
	BallControlFB.BallControl->STS.Disabled = 0;

	FB_BallControl(&BallControlFB);

	TEST_ASSERT_EQUAL_INT(STATE_STOPPING, BallControlFB.BallControl->STS.StateInt);

	TEST_DONE;
}

_TEST Test_Stopping_TransitionsToDisabled_WhenDisabledTrue(void)
{
	BallControlFB.BallControl->STS.StateInt = STATE_STOPPING;
	BallControlFB.BallControl->STS.Disabled = 1;

	FB_BallControl(&BallControlFB);

	TEST_ASSERT_EQUAL_INT(STATE_DISABLED, BallControlFB.BallControl->STS.StateInt);

	TEST_DONE;
}
/*
B+R UnitTest: This is generated code.
Do not edit! Do not move!
Description: UnitTest Testprogramm infrastructure (TestSet).
LastUpdated: 2026-05-07 12:33:52Z
By B+R UnitTest Helper Version: 2.0.2.35
*/
UNITTEST_FIXTURES(fixtures)
{
	new_TestFixture("Test_Stopping_StaysInStopping_WhenNotDisabled", Test_Stopping_StaysInStopping_WhenNotDisabled),
	new_TestFixture("Test_Stopping_TransitionsToDisabled_WhenDisabledTrue", Test_Stopping_TransitionsToDisabled_WhenDisabledTrue),
};

UNITTEST_CALLER_COMPLETE_EXPLICIT(testSet_BallControl_Stopping, "testSet_BallControl_Stopping", setupTest, 0, fixtures, 0, 0, 0);
```

### Program Logical/UnitTests/UnitTests/Tests_DistanceSensor_C (ANSIC)

#### variables.var - Name the suite and add PVs for the program
```iecst
(********************************************************************
 * COPYRIGHT --  MyAutomation-IT
 ********************************************************************
 * Program: Tests_DistanceSensor_C
 * File: variables.var
 * Author: Raivo Berends
 ********************************************************************
 * Local variables of program Tests_DistanceSensor_C
 ********************************************************************)
(*Describe the test*)
VAR
	Testsuite : UtMgrTestSuite := (Name:='DistanceSensor_Tests',Type:=utMgrTEST_TYPE_C);
END_VAR
(*Variables used in the tests*)
VAR
	DistanceSensorFB : FB_DistanceSensor;
	DistanceSensorStruct : UDT_DistanceSensor;
END_VAR
```

#### autoGeneratedFile.c - Auto generated code - list of all test sets in the program
```c
/*
B+R UnitTest: This is generated code.
Do not edit! Do not move!
Description: UnitTest Testprogramm infrastructure (List of TestSets).
LastUpdated: 2026-05-07 10:39:43Z
By B+R UnitTest Helper Version: 2.0.2.35
*/
#include "UnitTest.h"

UNITTEST_TESTSET_DECLARATION  testSet_DistanceSensor;

UNITTEST_TESTSET_FIXTURES(utTestSets)
{
	new_TestSet(testSet_DistanceSensor),
};
UNTITTEST_TESTSET_HANDLER();
```

#### testSet_DistanceSensor.c
```c
/********************************************************************
 * COPYRIGHT - MyAutoMation-IT
 ********************************************************************
 * Author: Raivo Berends
 ********************************************************************/

#include <bur/plctypes.h>

#ifdef _DEFAULT_INCLUDES
#include <AsDefault.h>
#endif

#include "UnitTest.h"
#include "Library.h"
#include "CommonTypes.h"
#include <string.h>

_SETUP_TEST(void)
{
	DistanceSensorFB.DistanceSensorLeft = &DistanceSensorStruct;
	DistanceSensorFB.DistanceSensorMiddle = &DistanceSensorStruct;
	DistanceSensorFB.DistanceSensorRight = &DistanceSensorStruct;

	memset(	DistanceSensorFB.DistanceSensorMiddle, 0, sizeof(*DistanceSensorFB.DistanceSensorMiddle));

	TEST_DONE;
}

_TEST Test_DistanceSensor_CombinesMSB_LSB(void)
{
	DistanceSensorFB.DistanceSensorMiddle->IO.DataLSB = BALL_MIN_DISTANCE + 100;

	FB_DistanceSensor(&DistanceSensorFB);

	TEST_ASSERT_EQUAL_INT(BALL_MIN_DISTANCE + 100, DistanceSensorFB.DistanceSensorMiddle->STS.Distance);

	TEST_DONE;
}

_TEST Test_DistanceSensor_ClampsOverloadToZero(void)
{
	DistanceSensorFB.DistanceSensorMiddle->IO.DataMSB = (OVERLOAD >> 8);
	DistanceSensorFB.DistanceSensorMiddle->IO.DataLSB = (OVERLOAD & 0xFF);

	FB_DistanceSensor(&DistanceSensorFB);

	TEST_ASSERT_EQUAL_INT(0, DistanceSensorFB.DistanceSensorMiddle->STS.Distance);

	TEST_DONE;
}

_TEST Test_DistanceSensor_ClampsUnderloadToZero(void)
{
	DistanceSensorFB.DistanceSensorMiddle->IO.DataMSB = (UNDERLOAD >> 8);
	DistanceSensorFB.DistanceSensorMiddle->IO.DataLSB = (UNDERLOAD & 0xFF);

	FB_DistanceSensor(&DistanceSensorFB);

	TEST_ASSERT_EQUAL_INT(0, DistanceSensorFB.DistanceSensorMiddle->STS.Distance);

	TEST_DONE;
}

_TEST Test_DistanceSensor_Out1BitMapping(void)
{
	DistanceSensorFB.DistanceSensorMiddle->IO.SensorInfo = OUT1_BITMASK;

	FB_DistanceSensor(&DistanceSensorFB);

	TEST_ASSERT_EQUAL_INT(OUT1_BITMASK, DistanceSensorFB.DistanceSensorMiddle->IO.OUT1);

	TEST_DONE;
}

_TEST Test_DistanceSensor_Out2BitMapping(void)
{
	DistanceSensorFB.DistanceSensorMiddle->IO.SensorInfo = OUT2_BITMASK;

	FB_DistanceSensor(&DistanceSensorFB);

	TEST_ASSERT_EQUAL_INT(1, DistanceSensorFB.DistanceSensorMiddle->IO.OUT2);

	TEST_DONE;
}

_TEST Test_DistanceSensor_DeviceStatusMapping(void)
{
	DistanceSensorFB.DistanceSensorMiddle->IO.SensorInfo = SENSOR_FAILURE << 4;

	FB_DistanceSensor(&DistanceSensorFB);

	TEST_ASSERT_EQUAL_INT(SENSOR_FAILURE, DistanceSensorFB.DistanceSensorMiddle->STS.DeviceStatus);

	TEST_DONE;
}

_TEST Test_DistanceSensor_BallDetectedInsideRange(void)
{
	DistanceSensorFB.DistanceSensorMiddle->IO.DataMSB = 0;
	DistanceSensorFB.DistanceSensorMiddle->IO.DataLSB = BALL_MIN_DISTANCE + 10;

	FB_DistanceSensor(&DistanceSensorFB);

	TEST_ASSERT_EQUAL_INT(60, DistanceSensorFB.DistanceSensorMiddle->STS.Distance);
	TEST_ASSERT_EQUAL_INT(1, DistanceSensorFB.DistanceSensorMiddle->STS.BallDetected);

	TEST_DONE;
}

_TEST Test_DistanceSensor_BallDetectedOutsideRange(void)
{
	DistanceSensorFB.DistanceSensorMiddle->STS.Distance = BALL_MAX_DISTANCE + 10;

	FB_DistanceSensor(&DistanceSensorFB);

	TEST_ASSERT_EQUAL_INT(0, DistanceSensorFB.DistanceSensorMiddle->STS.BallDetected);

	TEST_DONE;
}

_TEST Test_DistanceSensor_TooFarCondition(void)
{
	DistanceSensorFB.DistanceSensorMiddle->IO.DataMSB = 0x01;
	DistanceSensorFB.DistanceSensorMiddle->IO.DataLSB = 0x5E;

	FB_DistanceSensor(&DistanceSensorFB);

	TEST_ASSERT_EQUAL_INT(1, DistanceSensorFB.DistanceSensorMiddle->STS.TooFar);
	TEST_ASSERT_EQUAL_INT(1, DistanceSensorFB.DistanceSensorMiddle->ALM.OutOfBounds);

	TEST_DONE;
}

_TEST Test_DistanceSensor_TooCloseCondition(void)
{
	DistanceSensorFB.DistanceSensorMiddle->IO.DataMSB = 0;
	DistanceSensorFB.DistanceSensorMiddle->IO.DataLSB = 30;

	FB_DistanceSensor(&DistanceSensorFB);

	TEST_ASSERT_EQUAL_INT(1, DistanceSensorFB.DistanceSensorMiddle->STS.TooClose);
	TEST_ASSERT_EQUAL_INT(1, DistanceSensorFB.DistanceSensorMiddle->ALM.OutOfBounds);

	TEST_DONE;
}

_TEST Test_DistanceSensor_NormalRangeClearsFlags(void)
{
	DistanceSensorFB.DistanceSensorMiddle->IO.DataLSB = BALL_MIN_DISTANCE + 10;

	FB_DistanceSensor(&DistanceSensorFB);

	TEST_ASSERT_EQUAL_INT(0, DistanceSensorFB.DistanceSensorMiddle->STS.TooClose);
	TEST_ASSERT_EQUAL_INT(0, DistanceSensorFB.DistanceSensorMiddle->STS.TooFar);
	TEST_ASSERT_EQUAL_INT(0, DistanceSensorFB.DistanceSensorMiddle->ALM.OutOfBounds);

	TEST_DONE;
}

_TEST Test_DistanceSensor_DeviceFailureSetsAlarm(void)
{
	DistanceSensorFB.DistanceSensorMiddle->IO.SensorInfo = SENSOR_FAILURE << 4;

	FB_DistanceSensor(&DistanceSensorFB);

	TEST_ASSERT_EQUAL_INT(1, DistanceSensorFB.DistanceSensorMiddle->STS.AlarmActive);

	TEST_DONE;
}

_TEST Test_DistanceSensor_OutOfBoundsSetsAlarm(void)
{
	DistanceSensorFB.DistanceSensorMiddle->IO.DataMSB = 0x01;
	DistanceSensorFB.DistanceSensorMiddle->IO.DataLSB = 0x5E;

	FB_DistanceSensor(&DistanceSensorFB);

	TEST_ASSERT_EQUAL_INT(1, DistanceSensorFB.DistanceSensorMiddle->STS.AlarmActive);

	TEST_DONE;
}

_TEST Test_DistanceSensor_DeviceStatusZeroClearsAlarm(void)
{
	DistanceSensorFB.DistanceSensorMiddle->IO.DataLSB = BALL_MIN_DISTANCE;
	DistanceSensorFB.DistanceSensorMiddle->IO.SensorInfo = 0;

	FB_DistanceSensor(&DistanceSensorFB);

	TEST_ASSERT_EQUAL_INT(0, DistanceSensorFB.DistanceSensorMiddle->STS.AlarmActive);

	TEST_DONE;
}

_TEST Test_DistanceSensor_AlarmColourRed(void)
{
	DistanceSensorFB.DistanceSensorMiddle->STS.AlarmActive = 1;
	DistanceSensorFB.DistanceSensorMiddle->IO.SensorInfo = 0x40;

	FB_DistanceSensor(&DistanceSensorFB);

	TEST_ASSERT_EQUAL_INT(RED_COLOUR, DistanceSensorFB.DistanceSensorMiddle->STS.AlarmActiveColour);

	TEST_DONE;
}

_TEST Test_DistanceSensor_AlarmColourGreen(void)
{
	DistanceSensorFB.DistanceSensorMiddle->IO.DataLSB = BALL_MIN_DISTANCE + 10;
	DistanceSensorFB.DistanceSensorMiddle->STS.AlarmActive = 0;

	FB_DistanceSensor(&DistanceSensorFB);

	TEST_ASSERT_EQUAL_INT(GREEN_COLOUR, DistanceSensorFB.DistanceSensorMiddle->STS.AlarmActiveColour);

	TEST_DONE;
}

/*
B+R UnitTest: This is generated code.
Do not edit! Do not move!
Description: UnitTest Testprogramm infrastructure (TestSet).
LastUpdated: 2026-05-07 10:39:43Z
By B+R UnitTest Helper Version: 2.0.2.35
*/
UNITTEST_FIXTURES(fixtures)
{
	new_TestFixture("Test_DistanceSensor_CombinesMSB_LSB", Test_DistanceSensor_CombinesMSB_LSB),
	new_TestFixture("Test_DistanceSensor_ClampsOverloadToZero", Test_DistanceSensor_ClampsOverloadToZero),
	new_TestFixture("Test_DistanceSensor_ClampsUnderloadToZero", Test_DistanceSensor_ClampsUnderloadToZero),
	new_TestFixture("Test_DistanceSensor_Out1BitMapping", Test_DistanceSensor_Out1BitMapping),
	new_TestFixture("Test_DistanceSensor_Out2BitMapping", Test_DistanceSensor_Out2BitMapping),
	new_TestFixture("Test_DistanceSensor_DeviceStatusMapping", Test_DistanceSensor_DeviceStatusMapping),
	new_TestFixture("Test_DistanceSensor_BallDetectedInsideRange", Test_DistanceSensor_BallDetectedInsideRange),
	new_TestFixture("Test_DistanceSensor_BallDetectedOutsideRange", Test_DistanceSensor_BallDetectedOutsideRange),
	new_TestFixture("Test_DistanceSensor_TooFarCondition", Test_DistanceSensor_TooFarCondition),
	new_TestFixture("Test_DistanceSensor_TooCloseCondition", Test_DistanceSensor_TooCloseCondition),
	new_TestFixture("Test_DistanceSensor_NormalRangeClearsFlags", Test_DistanceSensor_NormalRangeClearsFlags),
	new_TestFixture("Test_DistanceSensor_DeviceFailureSetsAlarm", Test_DistanceSensor_DeviceFailureSetsAlarm),
	new_TestFixture("Test_DistanceSensor_OutOfBoundsSetsAlarm", Test_DistanceSensor_OutOfBoundsSetsAlarm),
	new_TestFixture("Test_DistanceSensor_DeviceStatusZeroClearsAlarm", Test_DistanceSensor_DeviceStatusZeroClearsAlarm),
	new_TestFixture("Test_DistanceSensor_AlarmColourRed", Test_DistanceSensor_AlarmColourRed),
	new_TestFixture("Test_DistanceSensor_AlarmColourGreen", Test_DistanceSensor_AlarmColourGreen),
};

UNITTEST_CALLER_COMPLETE_EXPLICIT(testSet_DistanceSensor, "testSet_DistanceSensor", setupTest, 0, fixtures, 0, 0, 0);
```

### Program Logical/UnitTests/UnitTests/Tests_FieldControl_C (ANSIC)

#### variables.var - Name the suite and add PVs for the program
```iecst
(********************************************************************
 * COPYRIGHT --  MyAutomation-IT
 ********************************************************************
 * Program: Tests_FieldControl_C
 * File: variables.var
 * Author: Raivo Berends
 ********************************************************************
 * Local variables of program Tests_FieldControl_C
 ********************************************************************)
(*Describe the test*)
VAR
	Testsuite : UtMgrTestSuite := (Name:='FieldControl_Tests',Type:=utMgrTEST_TYPE_C);
END_VAR
(*Variables used in the tests*)
VAR
	FieldControlFB : FB_FieldControl;
	FieldControlStruct : UDT_FieldControl;
	FieldMotorStruct : UDT_FieldMotor;
	InclinoSensorStruct : UDT_InclinoSensor;
END_VAR
```

#### autoGeneratedFile.c - Auto generated code - list of all test sets in the program
```c
/*
B+R UnitTest: This is generated code.
Do not edit! Do not move!
Description: UnitTest Testprogramm infrastructure (List of TestSets).
LastUpdated: 2026-05-07 13:11:07Z
By B+R UnitTest Helper Version: 2.0.2.35
*/
#include "UnitTest.h"

UNITTEST_TESTSET_DECLARATION  testSet_FieldControl_Disabled;
UNITTEST_TESTSET_DECLARATION  testSet_FieldControl_Initializing;
UNITTEST_TESTSET_DECLARATION  testSet_FieldControl_Idle;
UNITTEST_TESTSET_DECLARATION  testSet_FieldControl_Running;
UNITTEST_TESTSET_DECLARATION  testSet_FieldControl_Stopping;

UNITTEST_TESTSET_FIXTURES(utTestSets)
{
	new_TestSet(testSet_FieldControl_Disabled),
	new_TestSet(testSet_FieldControl_Initializing),
	new_TestSet(testSet_FieldControl_Idle),
	new_TestSet(testSet_FieldControl_Running),
	new_TestSet(testSet_FieldControl_Stopping),
};
UNTITTEST_TESTSET_HANDLER();
```

#### testSet_FieldControl_Disabled.c
```c
/********************************************************************
 * COPYRIGHT - MyAutoMation-IT
 ********************************************************************
 * Author: Raivo Berends
 ********************************************************************/

#include <bur/plctypes.h>

#ifdef _DEFAULT_INCLUDES
#include <AsDefault.h>
#endif

#include "UnitTest.h"
#include "Library.h"
#include "CommonTypes.h"
#include <string.h>

_SETUP_TEST(void)
{
	FieldControlFB.FieldControl = &FieldControlStruct;
	FieldControlFB.FieldMotor = &FieldMotorStruct;
	FieldControlFB.InclinoSensor = &InclinoSensorStruct;

	memset(FieldControlFB.FieldControl, 0, sizeof(*FieldControlFB.FieldControl));
	memset(FieldControlFB.FieldMotor, 0, sizeof(*FieldControlFB.FieldMotor));
	memset(FieldControlFB.InclinoSensor, 0, sizeof(*FieldControlFB.InclinoSensor));

	FieldControlFB.FieldControl->STS.StateInt = STATE_DISABLED;

	TEST_DONE;
}

_TEST Test_Disabled_ResetsAtTargetPosition(void)
{
	FieldControlFB.FieldControl->STS.AtTargetPosition = 1;

	FB_FieldControl(&FieldControlFB);

	TEST_ASSERT_EQUAL_INT(0, FieldControlFB.FieldControl->STS.AtTargetPosition);

	TEST_DONE;
}

_TEST Test_Disabled_IncreaseAngle_IncreasesAngle(void)
{
	FieldControlFB.FieldControl->PAR.Angle = 10.0;
	FieldControlFB.FieldControl->HMI.IncreaseAngle = 1;

	FB_FieldControl(&FieldControlFB);

	TEST_ASSERT_REAL_WITHIN(0.0001, 10.002, FieldControlFB.FieldControl->PAR.Angle);

	TEST_DONE;
}

_TEST Test_Disabled_IncreaseAngle_DoesNotExceedMax(void)
{
	FieldControlFB.FieldControl->PAR.Angle = MAX_ANGLE;
	FieldControlFB.FieldControl->HMI.IncreaseAngle = 1;

	FB_FieldControl(&FieldControlFB);

	TEST_ASSERT_EQUAL_DOUBLE(MAX_ANGLE, FieldControlFB.FieldControl->PAR.Angle);

	TEST_DONE;
}

_TEST Test_Disabled_DecreaseAngle_DecreasesAngle(void)
{
	FieldControlFB.FieldControl->PAR.Angle = 10.0;
	FieldControlFB.FieldControl->HMI.DecreaseAngle = 1;

	FB_FieldControl(&FieldControlFB);

	TEST_ASSERT_REAL_WITHIN(0.0001, 9.998, FieldControlFB.FieldControl->PAR.Angle);

	TEST_DONE;
}

_TEST Test_Disabled_DecreaseAngle_DoesNotGoBelowMin(void)
{
	FieldControlFB.FieldControl->PAR.Angle = MIN_ANGLE;
	FieldControlFB.FieldControl->HMI.DecreaseAngle = 1;

	FB_FieldControl(&FieldControlFB);

	TEST_ASSERT_EQUAL_DOUBLE(MIN_ANGLE, FieldControlFB.FieldControl->PAR.Angle);

	TEST_DONE;
}

_TEST Test_Disabled_TransitionsToInitializing(void)
{
	FieldControlFB.FieldControl->STS.Initializing = 1;

	FB_FieldControl(&FieldControlFB);

	TEST_ASSERT_EQUAL_INT(STATE_INITIALIZING, FieldControlFB.FieldControl->STS.StateInt);

	TEST_DONE;
}

_TEST Test_Disabled_StaysDisabled_WhenNotInitializing(void)
{
	FieldControlFB.FieldControl->STS.Initializing = 0;

	FB_FieldControl(&FieldControlFB);

	TEST_ASSERT_EQUAL_INT(STATE_DISABLED, FieldControlFB.FieldControl->STS.StateInt);

	TEST_DONE;
}

_TEST Test_Disabled_IncreaseHasPriorityOverDecrease(void)
{
	FieldControlFB.FieldControl->PAR.Angle = 10.0;

	FieldControlFB.FieldControl->HMI.IncreaseAngle = 1;
	FieldControlFB.FieldControl->HMI.DecreaseAngle = 1;

	FB_FieldControl(&FieldControlFB);

	TEST_ASSERT_REAL_WITHIN(0.0001, 10.002, FieldControlFB.FieldControl->PAR.Angle);

	TEST_DONE;
}
/*
B+R UnitTest: This is generated code.
Do not edit! Do not move!
Description: UnitTest Testprogramm infrastructure (TestSet).
LastUpdated: 2026-05-07 12:58:24Z
By B+R UnitTest Helper Version: 2.0.2.35
*/
UNITTEST_FIXTURES(fixtures)
{
	new_TestFixture("Test_Disabled_ResetsAtTargetPosition", Test_Disabled_ResetsAtTargetPosition),
	new_TestFixture("Test_Disabled_IncreaseAngle_IncreasesAngle", Test_Disabled_IncreaseAngle_IncreasesAngle),
	new_TestFixture("Test_Disabled_IncreaseAngle_DoesNotExceedMax", Test_Disabled_IncreaseAngle_DoesNotExceedMax),
	new_TestFixture("Test_Disabled_DecreaseAngle_DecreasesAngle", Test_Disabled_DecreaseAngle_DecreasesAngle),
	new_TestFixture("Test_Disabled_DecreaseAngle_DoesNotGoBelowMin", Test_Disabled_DecreaseAngle_DoesNotGoBelowMin),
	new_TestFixture("Test_Disabled_TransitionsToInitializing", Test_Disabled_TransitionsToInitializing),
	new_TestFixture("Test_Disabled_StaysDisabled_WhenNotInitializing", Test_Disabled_StaysDisabled_WhenNotInitializing),
	new_TestFixture("Test_Disabled_IncreaseHasPriorityOverDecrease", Test_Disabled_IncreaseHasPriorityOverDecrease),
};

UNITTEST_CALLER_COMPLETE_EXPLICIT(testSet_FieldControl_Disabled, "testSet_FieldControl_Disabled", setupTest, 0, fixtures, 0, 0, 0);
```

#### testSet_FieldControl_Initializing.c
```c
/********************************************************************
 * COPYRIGHT - MyAutoMation-IT
 ********************************************************************
 * Author: Raivo Berends
 ********************************************************************/

#include <bur/plctypes.h>

#ifdef _DEFAULT_INCLUDES
#include <AsDefault.h>
#endif

#include "UnitTest.h"
#include "Library.h"
#include "CommonTypes.h"
#include <string.h>

_SETUP_TEST(void)
{
	FieldControlFB.FieldControl = &FieldControlStruct;
	FieldControlFB.FieldMotor = &FieldMotorStruct;
	FieldControlFB.InclinoSensor = &InclinoSensorStruct;

	memset(FieldControlFB.FieldControl, 0, sizeof(*FieldControlFB.FieldControl));
	memset(FieldControlFB.FieldMotor, 0, sizeof(*FieldControlFB.FieldMotor));
	memset(FieldControlFB.InclinoSensor, 0, sizeof(*FieldControlFB.InclinoSensor));

	FieldControlFB.FieldControl->STS.StateInt = STATE_INITIALIZING;

	TEST_DONE;
}

_TEST Test_Initializing_TransitionsToIdle(void)
{
	FieldControlFB.FieldControl->STS.Idle = 1;

	FB_FieldControl(&FieldControlFB);

	TEST_ASSERT_EQUAL_INT(STATE_IDLE, FieldControlFB.FieldControl->STS.StateInt);

	TEST_DONE;
}

_TEST Test_Initializing_SetsAtTargetPosition_WhenAligned(void)
{
	FieldControlFB.FieldControl->STS.Idle = 0;

	FieldControlFB.FieldControl->STS.CurrentAngle = 9.38;
	FieldControlFB.FieldControl->PAR.Angle = 10.0;

	FieldControlFB.FieldControl->STS.AtTargetPosition = 0;

	FieldControlFB.FieldMotor->STS.EndButtonHit = 1;

	FB_FieldControl(&FieldControlFB);

	TEST_ASSERT_EQUAL_INT(1, FieldControlFB.FieldControl->STS.AtTargetPosition);

	TEST_DONE;
}

_TEST Test_Initializing_DoesNotSetTarget_WhenAngleNotReached(void)
{
	FieldControlFB.FieldControl->STS.Idle = 0;

	FieldControlFB.FieldControl->STS.CurrentAngle = 1.0;
	FieldControlFB.FieldControl->PAR.Angle = 15.0;

	FieldControlFB.FieldControl->STS.AtTargetPosition = 0;

	FieldControlFB.FieldMotor->STS.EndButtonHit = 1;

	FB_FieldControl(&FieldControlFB);

	TEST_ASSERT_EQUAL_INT(0, FieldControlFB.FieldControl->STS.AtTargetPosition);

	TEST_DONE;
}

_TEST Test_Initializing_DoesNotSetTarget_WhenAlreadyAtTarget(void)
{
	FieldControlFB.FieldControl->STS.Idle = 0;

	FieldControlFB.FieldControl->STS.CurrentAngle = 10.0;
	FieldControlFB.FieldControl->PAR.Angle = 10.0;

	FieldControlFB.FieldControl->STS.AtTargetPosition = 1;

	FieldControlFB.FieldMotor->STS.EndButtonHit = 1;

	FB_FieldControl(&FieldControlFB);

	TEST_ASSERT_EQUAL_INT(1, FieldControlFB.FieldControl->STS.AtTargetPosition);

	TEST_DONE;
}

_TEST Test_Initializing_DoesNotSetTarget_WithoutEndButton(void)
{
	FieldControlFB.FieldControl->STS.Idle = 0;

	FieldControlFB.FieldControl->STS.CurrentAngle = 10.0;
	FieldControlFB.FieldControl->PAR.Angle = 10.0;

	FieldControlFB.FieldControl->STS.AtTargetPosition = 0;

	FieldControlFB.FieldMotor->STS.EndButtonHit = 0;

	FB_FieldControl(&FieldControlFB);

	TEST_ASSERT_EQUAL_INT(0, FieldControlFB.FieldControl->STS.AtTargetPosition);

	TEST_DONE;
}

_TEST Test_Initializing_IdleHasPriorityOverAlignment(void)
{
	FieldControlFB.FieldControl->STS.Idle = 1;

	FieldControlFB.FieldControl->STS.CurrentAngle = 10.0;
	FieldControlFB.FieldControl->PAR.Angle = 10.0;

	FieldControlFB.FieldControl->STS.AtTargetPosition = 0;

	FieldControlFB.FieldMotor->STS.EndButtonHit = 1;

	FB_FieldControl(&FieldControlFB);

	TEST_ASSERT_EQUAL_INT(STATE_IDLE, FieldControlFB.FieldControl->STS.StateInt);
	TEST_ASSERT_EQUAL_INT(0, FieldControlFB.FieldControl->STS.AtTargetPosition);

	TEST_DONE;
}
/*
B+R UnitTest: This is generated code.
Do not edit! Do not move!
Description: UnitTest Testprogramm infrastructure (TestSet).
LastUpdated: 2026-05-07 13:11:07Z
By B+R UnitTest Helper Version: 2.0.2.35
*/
UNITTEST_FIXTURES(fixtures)
{
	new_TestFixture("Test_Initializing_TransitionsToIdle", Test_Initializing_TransitionsToIdle),
	new_TestFixture("Test_Initializing_SetsAtTargetPosition_WhenAligned", Test_Initializing_SetsAtTargetPosition_WhenAligned),
	new_TestFixture("Test_Initializing_DoesNotSetTarget_WhenAngleNotReached", Test_Initializing_DoesNotSetTarget_WhenAngleNotReached),
	new_TestFixture("Test_Initializing_DoesNotSetTarget_WhenAlreadyAtTarget", Test_Initializing_DoesNotSetTarget_WhenAlreadyAtTarget),
	new_TestFixture("Test_Initializing_DoesNotSetTarget_WithoutEndButton", Test_Initializing_DoesNotSetTarget_WithoutEndButton),
	new_TestFixture("Test_Initializing_IdleHasPriorityOverAlignment", Test_Initializing_IdleHasPriorityOverAlignment),
};

UNITTEST_CALLER_COMPLETE_EXPLICIT(testSet_FieldControl_Initializing, "testSet_FieldControl_Initializing", setupTest, 0, fixtures, 0, 0, 0);
```
